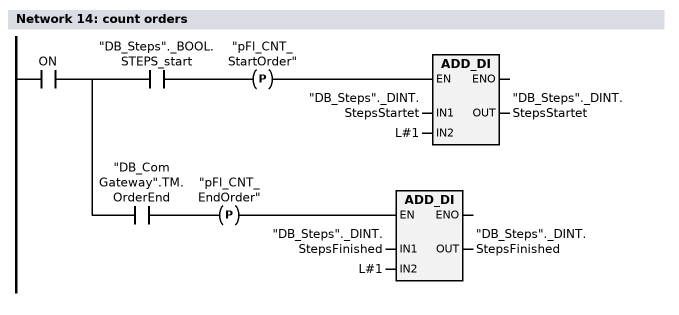
[picture p118: STEPS_OrderData networks 14-14]
NETWORK
TITLE = count orders
      A     "ON";
      =     L 35.0;
      A     L 35.0;
      A(;
      A     "DB_Steps"._BOOL.STEPS_start;
      BLD   100;
      FP    "pFl_CNT_StartOrder";
      );
      JNB   _007;
      L     "DB_Steps"._DINT.StepsStartet;
      L     L#1;
      +D;
      T     "DB_Steps"._DINT.StepsStartet;
_007: NOP   0;
      A     L 35.0;
      A(;
      A     "DB_ComGateway".TM.OrderEnd;
      BLD   100;
      FP    "pFl_CNT_EndOrder";
      );
      JNB   _008;
      L     "DB_Steps"._DINT.StepsFinished;
      L     L#1;
      +D;
      T     "DB_Steps"._DINT.StepsFinished;
_008: NOP   0;
END_FUNCTION

FUNCTION "STEPS_EMPTY" : VOID	// FC 113
TITLE = Steps Empty
VERSION : 0.1
BEGIN
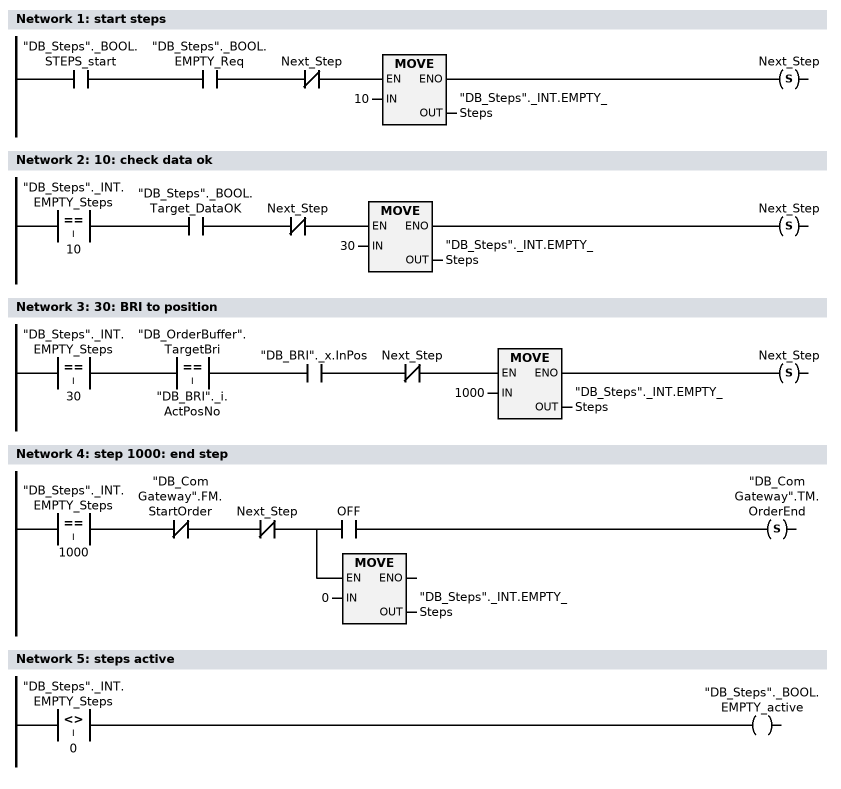
NETWORK
TITLE = start steps
      A     "DB_Steps"._BOOL.STEPS_start;
      A     "DB_Steps"._BOOL.EMPTY_Req;
      AN    "Next_Step";
      JNB   _001;
      L     10;
      T     "DB_Steps"._INT.EMPTY_Steps;
      SET;
      SAVE;
      CLR;
_001: A     BR;
      S     "Next_Step";
NETWORK
TITLE = 10: check data ok
      A(;
      L     "DB_Steps"._INT.EMPTY_Steps;
      L     10;
      ==I;
      );
      A     "DB_Steps"._BOOL.Target_DataOK;
      AN    "Next_Step";
      JNB   _002;
      L     30;
      T     "DB_Steps"._INT.EMPTY_Steps;
      SET;
      SAVE;
      CLR;
_002: A     BR;
      S     "Next_Step";
NETWORK
TITLE = 30: BRI to position
//1000: end of steps
      A(;
      L     "DB_Steps"._INT.EMPTY_Steps;
      L     30;
      ==I;
      );
      A(;
      L     "DB_OrderBuffer".TargetBri;
      L     "DB_BRI"._i.ActPosNo;
      ==I;
      );
      A     "DB_BRI"._x.InPos;
      AN    "Next_Step";
      JNB   _003;
      L     1000;
      T     "DB_Steps"._INT.EMPTY_Steps;
      SET;
      SAVE;
      CLR;
_003: A     BR;
      S     "Next_Step";
NETWORK
TITLE = step 1000: end step
//because of time reason we disable the finish flag
//also we check at the end the start bit has been cleared
      A(;
      L     "DB_Steps"._INT.EMPTY_Steps;
      L     1000;
      ==I;
      );
      AN    "DB_ComGateway".FM.StartOrder;
      AN    "Next_Step";
      =     L 0.0;
      A     L 0.0;
      A     "OFF";
      S     "DB_ComGateway".TM.OrderEnd;
      A     L 0.0;
      JNB   _004;
      L     0;
      T     "DB_Steps"._INT.EMPTY_Steps;
_004: NOP   0;
NETWORK
TITLE = steps active
      L     "DB_Steps"._INT.EMPTY_Steps;
      L     0;
      <>I;
      =     "DB_Steps"._BOOL.EMPTY_active;
END_FUNCTION

FUNCTION "Axis_BRIDGE" : VOID	// FC 200
TITLE = Axis BRIDGE
AUTHOR : Koenig
VERSION : 0.1
VAR_TEMP
  Signal : BOOL ;
  TEMP_01 : BOOL ;
  TEMP_02 : BOOL ;
  Encoder : DINT ;
  Temp_Dint : DINT ;
END_VAR
BEGIN
NETWORK
TITLE =
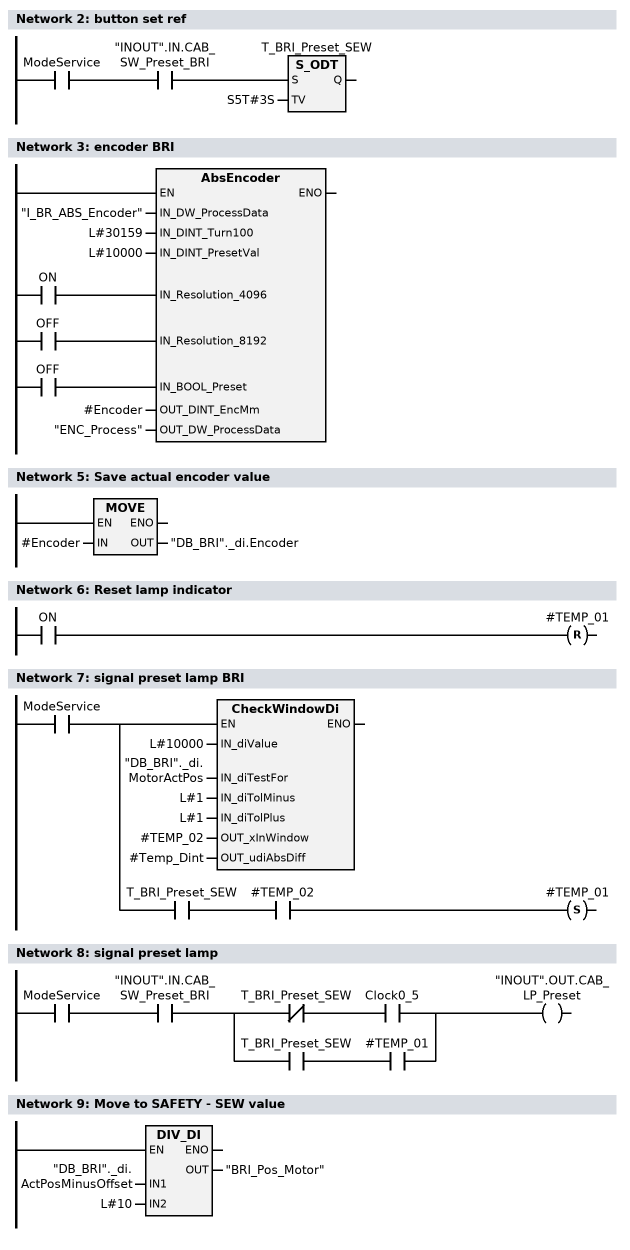
NETWORK
TITLE = button set ref
      A     "ModeService";
      A     "INOUT".IN.CAB_SW_Preset_BRI;
      L     S5T#3S;
      SD    "T_BRI_Preset_SEW";
      NOP   0;
      NOP   0;
      NOP   0;
      NOP   0;
NETWORK
TITLE = encoder BRI
      A     "ON";
      =     L 10.0;
      BLD   103;
      A     "OFF";
      =     L 10.1;
      BLD   103;
      A     "OFF";
      =     L 10.2;
      BLD   103;
      CALL  "AbsEncoder" (
           IN_DW_ProcessData        := "I_BR_ABS_Encoder",
           IN_DINT_Turn100          := L#30159,
           IN_DINT_PresetVal        := L#10000,
           IN_Resolution_4096       := L 10.0,
           IN_Resolution_8192       := L 10.1,
           IN_BOOL_Preset           := L 10.2,
           OUT_DINT_EncMm           := #Encoder,
           OUT_DW_ProcessData       := "ENC_Process");
      NOP   0;
NETWORK
TITLE = Preset encoder T&R
      A     "T_BRI_Preset_SEW";
      =     L 10.0;
      BLD   103;
      BLD   9;
      =     L 15.0;
      CDB;
      OPN   DI 50;
      TAR2  LD 11;
      A     L 10.0;
      =     DIX 0.0;
      L     L#2038;
      T     DID 2;
      L     2;
      T     DIW 6;
      L     4;
      T     DIW 8;
      L     W#16#1002;
      T     DIW 16;
      L     4;
      T     DIW 18;
      L     0;
      T     DIW 20;
      L     P#M 84.0;
      T     DID 22;
      LAR2  P#DBX 0.0;
      UC    "WRREC";
      LAR2  LD 11;
      CDB;
      BLD   10;
      NOP   0;
NETWORK
TITLE = Save actual encoder value
      L     #Encoder;
      T     "DB_BRI"._di.Encoder;
      NOP   0;
NETWORK
TITLE = Reset lamp indicator
      A     "ON";
      R     #TEMP_01;
NETWORK
TITLE = signal preset lamp BRI
      A     "ModeService";
      =     L 10.0;
      A     L 10.0;
      JNB   _001;
      CALL  "CheckWindowDi" (
           IN_diValue               := L#10000,
           IN_diTestFor             := "DB_BRI"._di.MotorActPos,
           IN_diTolMinus            := L#1,
           IN_diTolPlus             := L#1,
           OUT_xInWindow            := #TEMP_02,
           OUT_udiAbsDiff           := #Temp_Dint);
_001: NOP   0;
      A     L 10.0;
      A     "T_BRI_Preset_SEW";
      A     #TEMP_02;
      S     #TEMP_01;
NETWORK
TITLE = signal preset lamp
      A     "ModeService";
      A     "INOUT".IN.CAB_SW_Preset_BRI;
      A(;
      AN    "T_BRI_Preset_SEW";
      A     "Clock0_5";
      O;
      A     "T_BRI_Preset_SEW";
      A     #TEMP_01;
      );
      =     "INOUT".OUT.CAB_LP_Preset;
NETWORK
TITLE = Move to SAFETY - SEW value
      L     "DB_BRI"._di.ActPosMinusOffset;
      L     L#10;
      /D;
      T     "BRI_Pos_Motor";
      NOP   0;
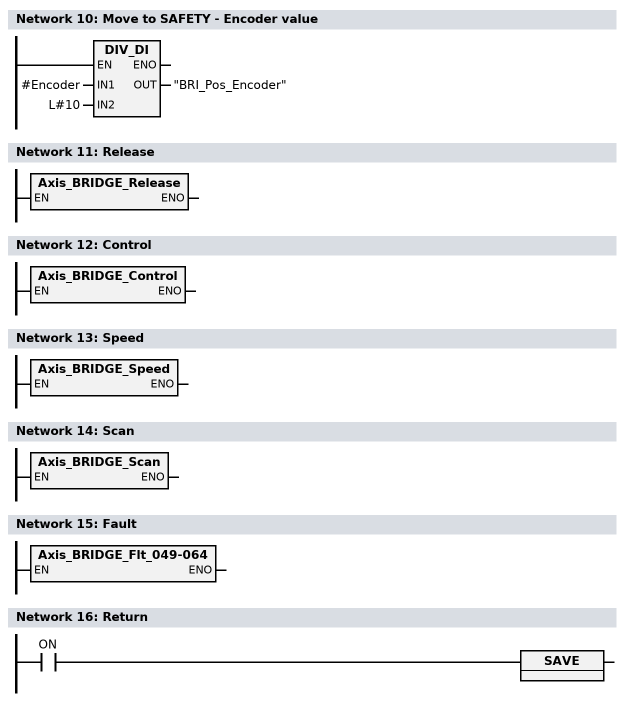
NETWORK
TITLE = Move to SAFETY - Encoder value
      L     #Encoder;
      L     L#10;
      /D;
      T     "BRI_Pos_Encoder";
      NOP   0;
NETWORK
TITLE = Release
      CALL  "Axis_BRIDGE_Release";
      NOP   0;
NETWORK
TITLE = Control
      CALL  "Axis_BRIDGE_Control";
      NOP   0;
NETWORK
TITLE = Speed
      CALL  "Axis_BRIDGE_Speed";
      NOP   0;
NETWORK
TITLE = Scan
      CALL  "Axis_BRIDGE_Scan";
      NOP   0;
NETWORK
TITLE = Fault
      CALL  "Axis_BRIDGE_Flt_049-064";
      NOP   0;
NETWORK
TITLE = Return
      A     "ON";
      SAVE;
END_FUNCTION

FUNCTION "Axis_BRIDGE_Release" : VOID	// FC 201
TITLE = Axis BRIDGE Release
VERSION : 0.1
BEGIN
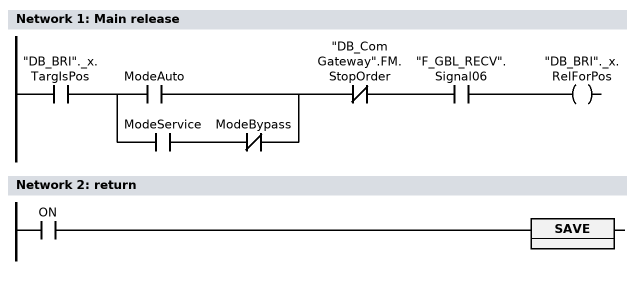
NETWORK
TITLE = Main release
      A     "DB_BRI"._x.TargIsPos;
      A(;
      O     "ModeAuto";
      O;
      A     "ModeService";
      AN    "ModeBypass";
      );
      AN    "DB_ComGateway".FM.StopOrder;
      A     "F_GBL_RECV".Signal06;
      =     "DB_BRI"._x.RelForPos;
NETWORK
TITLE = return
      A     "ON";
      SAVE;
END_FUNCTION

FUNCTION "Axis_BRIDGE_Control" : VOID	// FC 202
TITLE = BRIDGE Control
VERSION : 0.1
VAR_TEMP
  PositionMode : BOOL ;
  tmp_TagetPos_Auto : BOOL ;
  tmp_TagetPos_Manual : BOOL ;
  tmp_TargetValueOK : BOOL ;
  Mode_ref : BOOL ;
  Mode_jog : BOOL ;
  Error : WORD ;
  Next : DINT ;
  Prev : DINT ;
  First : DINT ;
  Last : DINT ;
END_VAR
BEGIN
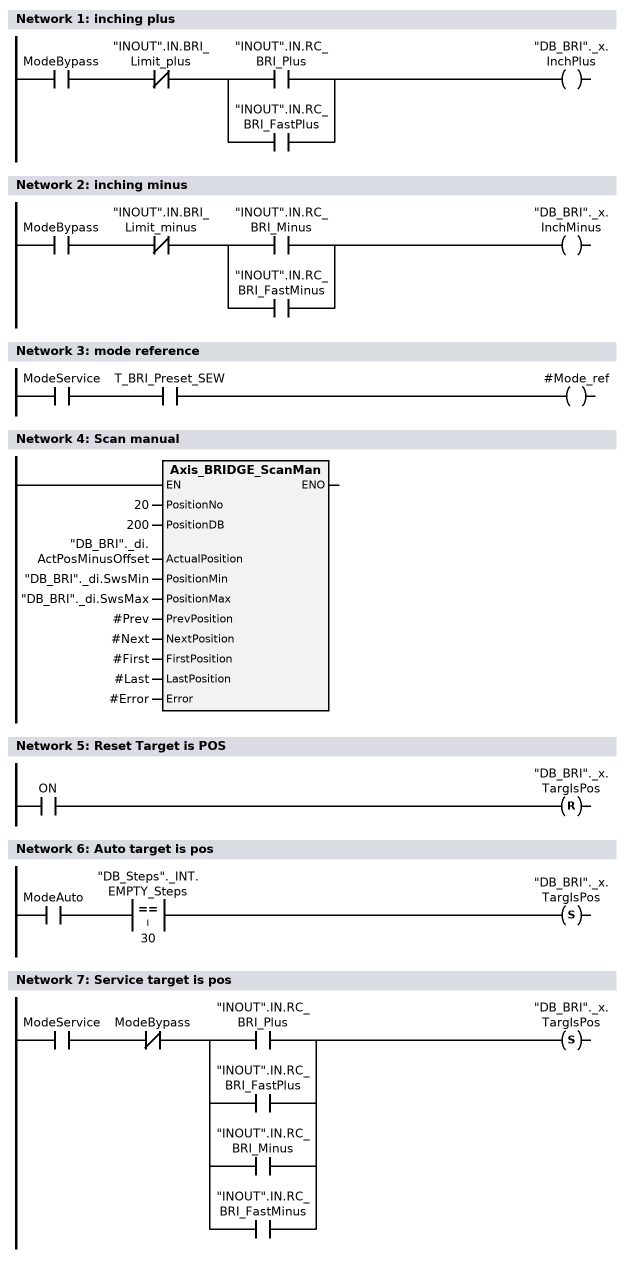
NETWORK
TITLE = inching plus
//in Service with bypass we use jog mode
      A     "ModeBypass";
      AN    "INOUT".IN.BRI_Limit_plus;
      A(;
      O     "INOUT".IN.RC_BRI_Plus;
      O     "INOUT".IN.RC_BRI_FastPlus;
      );
      =     "DB_BRI"._x.InchPlus;
NETWORK
TITLE = inching minus
      A     "ModeBypass";
      AN    "INOUT".IN.BRI_Limit_minus;
      A(;
      O     "INOUT".IN.RC_BRI_Minus;
      O     "INOUT".IN.RC_BRI_FastMinus;
      );
      =     "DB_BRI"._x.InchMinus;
NETWORK
TITLE = mode reference
      A     "ModeService";
      A     "T_BRI_Preset_SEW";
      =     #Mode_ref;
NETWORK
TITLE = Scan manual
      CALL  "Axis_BRIDGE_ScanMan" (
           PositionNo               := 20,
           PositionDB               := 200,
           ActualPosition           := "DB_BRI"._di.ActPosMinusOffset,
           PositionMin              := "DB_BRI"._di.SwsMin,
           PositionMax              := "DB_BRI"._di.SwsMax,
           PrevPosition             := #Prev,
           NextPosition             := #Next,
           FirstPosition            := #First,
           LastPosition             := #Last,
           Error                    := #Error);
      NOP   0;
NETWORK
TITLE = Reset Target is POS
      A     "ON";
      R     "DB_BRI"._x.TargIsPos;
NETWORK
TITLE = Auto target is pos
      A     "ModeAuto";
      A(;
      L     "DB_Steps"._INT.EMPTY_Steps;
      L     30;
      ==I;
      );
      S     "DB_BRI"._x.TargIsPos;
NETWORK
TITLE = Service target is pos
      A     "ModeService";
      AN    "ModeBypass";
      A(;
      O     "INOUT".IN.RC_BRI_Plus;
      O     "INOUT".IN.RC_BRI_FastPlus;
      O     "INOUT".IN.RC_BRI_Minus;
      O     "INOUT".IN.RC_BRI_FastMinus;
      );
      S     "DB_BRI"._x.TargIsPos;
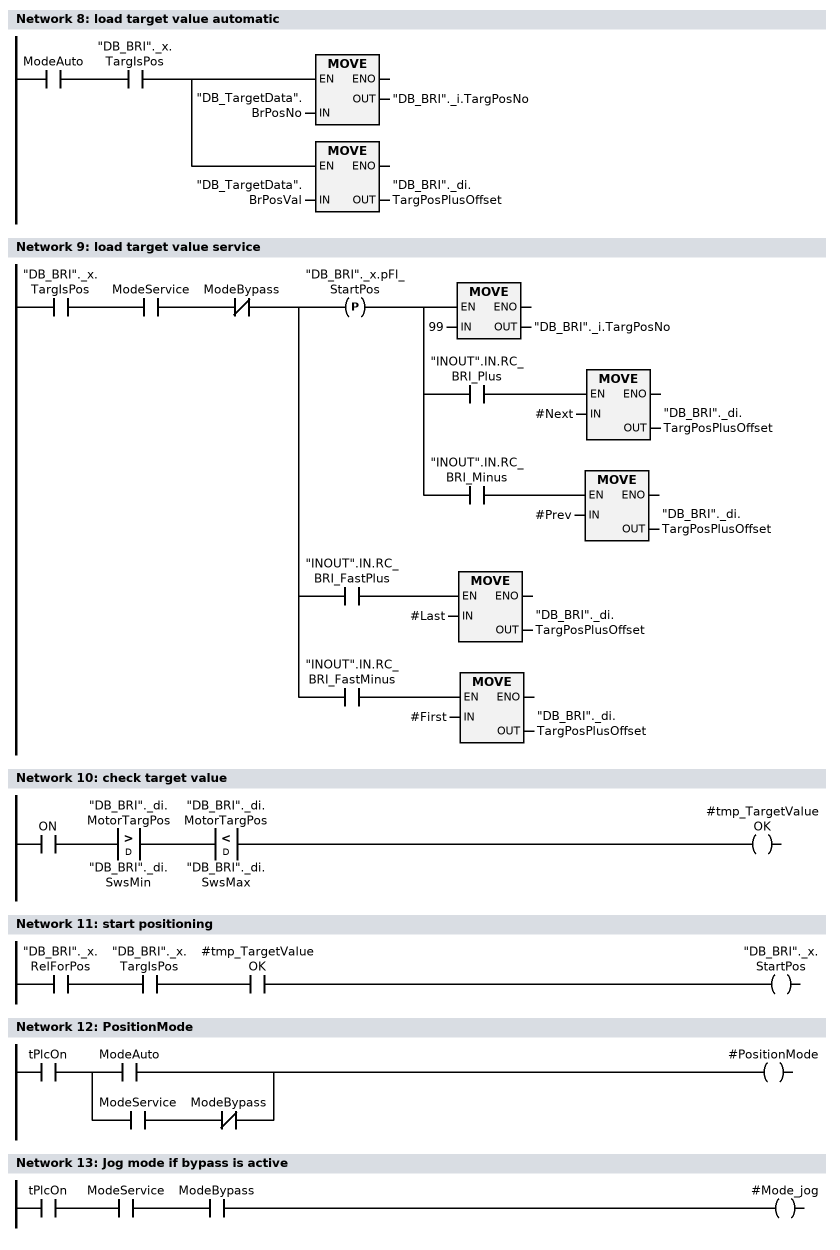
NETWORK
TITLE = load target value automatic
      A     "ModeAuto";
      A     "DB_BRI"._x.TargIsPos;
      =     L 20.0;
      A     L 20.0;
      JNB   _001;
      L     "DB_TargetData".BrPosNo;
      T     "DB_BRI"._i.TargPosNo;
_001: NOP   0;
      A     L 20.0;
      JNB   _002;
      L     "DB_TargetData".BrPosVal;
      T     "DB_BRI"._di.TargPosPlusOffset;
_002: NOP   0;
NETWORK
TITLE = load target value service
//In service we load the next/prev value or min/max
      A     "DB_BRI"._x.TargIsPos;
      A     "ModeService";
      AN    "ModeBypass";
      =     L 20.0;
      A     L 20.0;
      FP    "DB_BRI"._x.pFl_StartPos;
      =     L 20.1;
      A     L 20.1;
      JNB   _003;
      L     99;
      T     "DB_BRI"._i.TargPosNo;
_003: NOP   0;
      A     L 20.1;
      A     "INOUT".IN.RC_BRI_Plus;
      JNB   _004;
      L     #Next;
      T     "DB_BRI"._di.TargPosPlusOffset;
_004: NOP   0;
      A     L 20.1;
      A     "INOUT".IN.RC_BRI_Minus;
      JNB   _005;
      L     #Prev;
      T     "DB_BRI"._di.TargPosPlusOffset;
_005: NOP   0;
      A     L 20.0;
      A     "INOUT".IN.RC_BRI_FastPlus;
      JNB   _006;
      L     #Last;
      T     "DB_BRI"._di.TargPosPlusOffset;
_006: NOP   0;
      A     L 20.0;
      A     "INOUT".IN.RC_BRI_FastMinus;
      JNB   _007;
      L     #First;
      T     "DB_BRI"._di.TargPosPlusOffset;
_007: NOP   0;
NETWORK
TITLE = check target value
      A     "ON";
      A(;
      L     "DB_BRI"._di.MotorTargPos;
      L     "DB_BRI"._di.SwsMin;
      >D;
      );
      A(;
      L     "DB_BRI"._di.MotorTargPos;
      L     "DB_BRI"._di.SwsMax;
      <D;
      );
      =     #tmp_TargetValueOK;
NETWORK
TITLE = start positioning
      A     "DB_BRI"._x.RelForPos;
      A     "DB_BRI"._x.TargIsPos;
      A     #tmp_TargetValueOK;
      =     "DB_BRI"._x.StartPos;
NETWORK
TITLE = PositionMode
      A     "tPlcOn";
      A(;
      O     "ModeAuto";
      O;
      A     "ModeService";
      AN    "ModeBypass";
      );
      =     #PositionMode;
NETWORK
TITLE = Jog mode if bypass is active
      A     "tPlcOn";
      A     "ModeService";
      A     "ModeBypass";
      =     #Mode_jog;
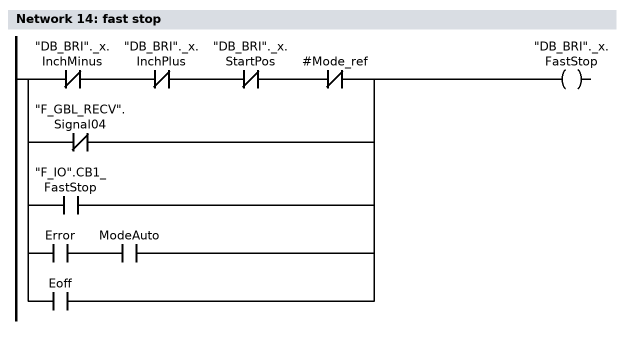
NETWORK
TITLE = fast stop
      AN    "DB_BRI"._x.InchMinus;
      AN    "DB_BRI"._x.InchPlus;
      AN    "DB_BRI"._x.StartPos;
      AN    #Mode_ref;
      ON    "F_GBL_RECV".Signal04;
      O     "F_IO".CB1_FastStop;
      O;
      A     "Error";
      A     "ModeAuto";
      O     "Eoff";
      =     "DB_BRI"._x.FastStop;
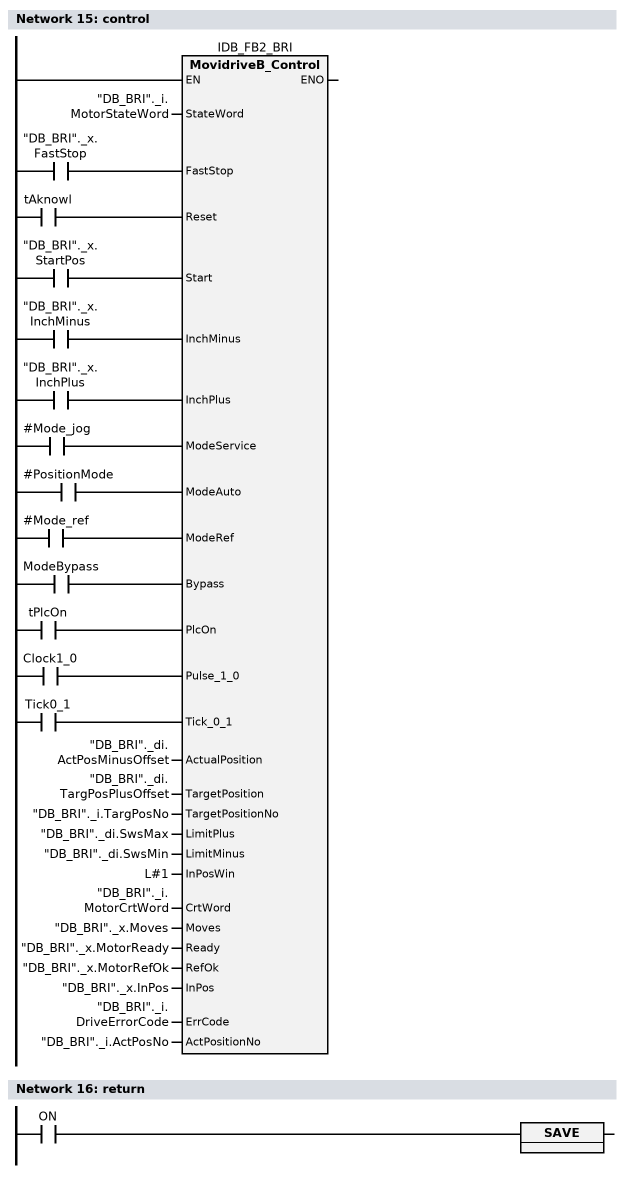
NETWORK
TITLE = control
      A     "DB_BRI"._x.FastStop;
      =     L 20.0;
      BLD   103;
      A     "tAknowl";
      =     L 20.1;
      BLD   103;
      A     "DB_BRI"._x.StartPos;
      =     L 20.2;
      BLD   103;
      A     "DB_BRI"._x.InchMinus;
      =     L 20.3;
      BLD   103;
      A     "DB_BRI"._x.InchPlus;
      =     L 20.4;
      BLD   103;
      A     #Mode_jog;
      =     L 20.5;
      BLD   103;
      A     #PositionMode;
      =     L 20.6;
      BLD   103;
      A     #Mode_ref;
      =     L 20.7;
      BLD   103;
      A     "ModeBypass";
      =     L 21.0;
      BLD   103;
      A     "tPlcOn";
      =     L 21.1;
      BLD   103;
      A     "Clock1_0";
      =     L 21.2;
      BLD   103;
      A     "Tick0_1";
      =     L 21.3;
      BLD   103;
      CALL  "MovidriveB_Control" , "IDB_FB2_BRI" (
           StateWord                := "DB_BRI"._i.MotorStateWord,
           FastStop                 := L 20.0,
           Reset                    := L 20.1,
           Start                    := L 20.2,
           InchMinus                := L 20.3,
           InchPlus                 := L 20.4,
           ModeService              := L 20.5,
           ModeAuto                 := L 20.6,
           ModeRef                  := L 20.7,
           Bypass                   := L 21.0,
           PlcOn                    := L 21.1,
           Pulse_1_0                := L 21.2,
           Tick_0_1                 := L 21.3,
           ActualPosition           := "DB_BRI"._di.ActPosMinusOffset,
           TargetPosition           := "DB_BRI"._di.TargPosPlusOffset,
           TargetPositionNo         := "DB_BRI"._i.TargPosNo,
           LimitPlus                := "DB_BRI"._di.SwsMax,
           LimitMinus               := "DB_BRI"._di.SwsMin,
           InPosWin                 := L#1,
           CrtWord                  := "DB_BRI"._i.MotorCrtWord,
           Moves                    := "DB_BRI"._x.Moves,
           Ready                    := "DB_BRI"._x.MotorReady,
           RefOk                    := "DB_BRI"._x.MotorRefOk,
           InPos                    := "DB_BRI"._x.InPos,
           ErrCode                  := "DB_BRI"._i.DriveErrorCode,
           ActPositionNo            := "DB_BRI"._i.ActPosNo);
      NOP   0;
NETWORK
TITLE = return
      A     "ON";
      SAVE;
END_FUNCTION

FUNCTION "Axis_BRIDGE_Speed" : VOID	// FC 203
TITLE = BRIDGE Speed
VERSION : 0.1
VAR_TEMP
  tmp_di_1 : DINT ;
  tmp_di_2 : DINT ;
  tmp_i_1 : INT ;
  tmp_i_2 : INT ;
  tmp_speed : INT ;
  tmp_diff_Pos : DINT ;
  tmp_Slow_Pos : BOOL ;
  tmp_Dcc : INT ;
END_VAR
BEGIN
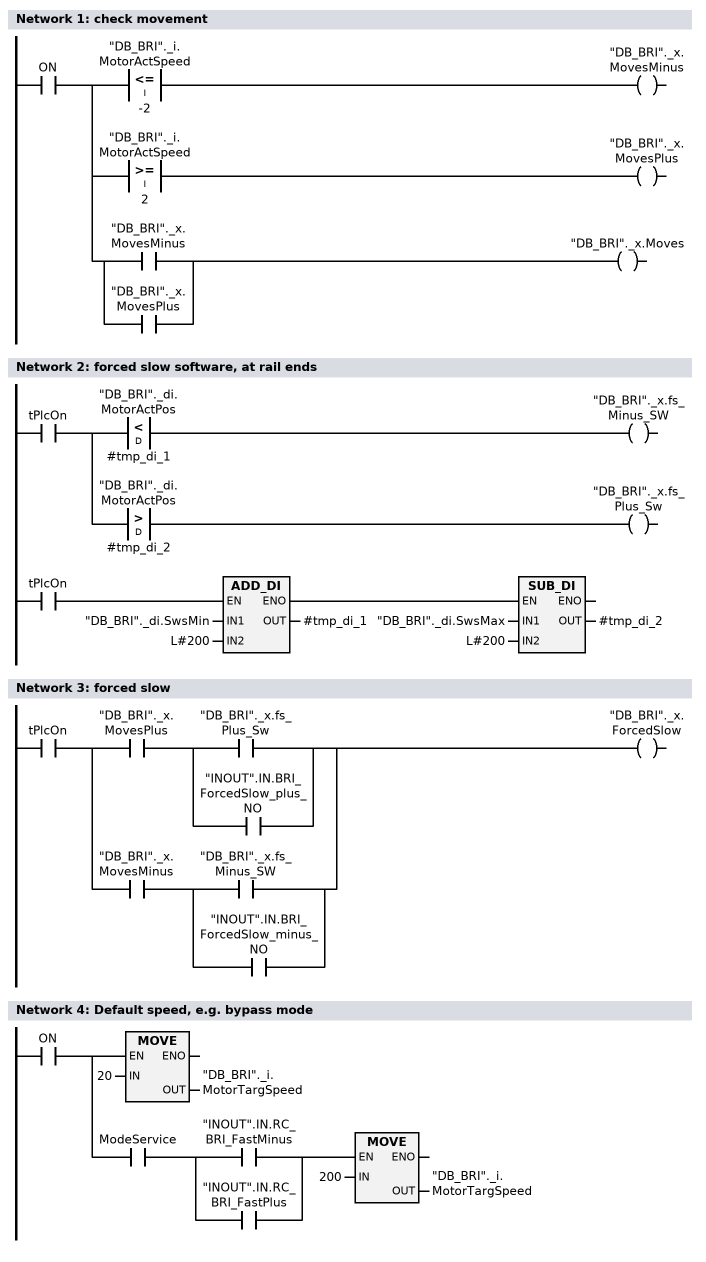
NETWORK
TITLE = check movement
      A     "ON";
      =     L 22.0;
      A     L 22.0;
      A(;
      L     "DB_BRI"._i.MotorActSpeed;
      L     -2;
      <=I;
      );
      =     "DB_BRI"._x.MovesMinus;
      A     L 22.0;
      A(;
      L     "DB_BRI"._i.MotorActSpeed;
      L     2;
      >=I;
      );
      =     "DB_BRI"._x.MovesPlus;
      A     L 22.0;
      A(;
      O     "DB_BRI"._x.MovesMinus;
      O     "DB_BRI"._x.MovesPlus;
      );
      =     "DB_BRI"._x.Moves;
NETWORK
TITLE = forced slow software, at rail ends
//Old distance: 1000mm
      A     "tPlcOn";
      =     L 22.0;
      A(;
      A     L 22.0;
      JNB   _001;
      L     "DB_BRI"._di.SwsMin;
      L     L#200;
      +D;
      T     #tmp_di_1;
      AN    OV;
      SAVE;
      CLR;
_001: A     BR;
      );
      JNB   _002;
      L     "DB_BRI"._di.SwsMax;
      L     L#200;
      -D;
      T     #tmp_di_2;
_002: NOP   0;
      A     L 22.0;
      A(;
      L     "DB_BRI"._di.MotorActPos;
      L     #tmp_di_1;
      <D;
      );
      =     "DB_BRI"._x.fs_Minus_SW;
      A     L 22.0;
      A(;
      L     "DB_BRI"._di.MotorActPos;
      L     #tmp_di_2;
      >D;
      );
      =     "DB_BRI"._x.fs_Plus_Sw;
NETWORK
TITLE = forced slow
//in service we use only the software, in auto we use the prox. switches
      A     "tPlcOn";
      A(;
      A     "DB_BRI"._x.MovesPlus;
      A(;
      O     "DB_BRI"._x.fs_Plus_Sw;
      O     "INOUT".IN.BRI_ForcedSlow_plus_NO;
      );
      O;
      A     "DB_BRI"._x.MovesMinus;
      A(;
      O     "DB_BRI"._x.fs_Minus_SW;
      O     "INOUT".IN.BRI_ForcedSlow_minus_NO;
      );
      );
      =     "DB_BRI"._x.ForcedSlow;
NETWORK
TITLE = Default speed, e.g. bypass mode
//in bypass we can also drive a little faster
//
      A     "ON";
      =     L 22.0;
      A     L 22.0;
      JNB   _003;
      L     20;
      T     "DB_BRI"._i.MotorTargSpeed;
_003: NOP   0;
      A     L 22.0;
      A     "ModeService";
      A(;
      O     "INOUT".IN.RC_BRI_FastMinus;
      O     "INOUT".IN.RC_BRI_FastPlus;
      );
      JNB   _004;
      L     200;
      T     "DB_BRI"._i.MotorTargSpeed;
_004: NOP   0;
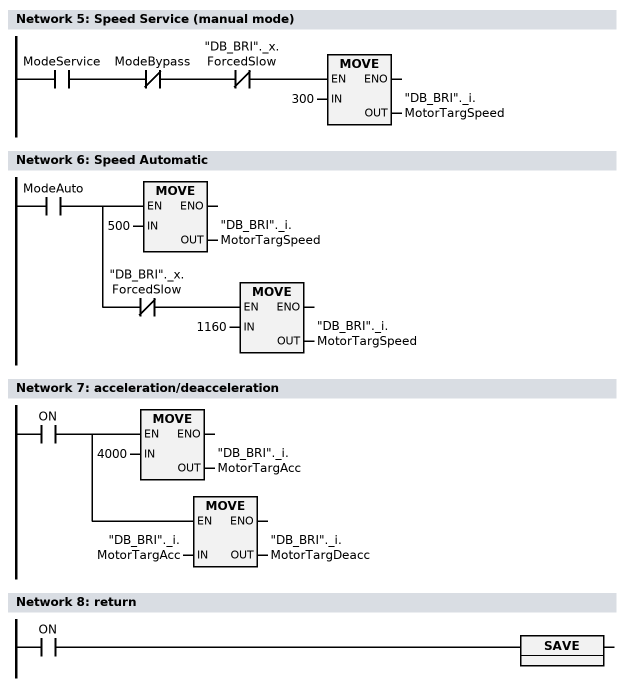
NETWORK
TITLE = Speed Service (manual mode)
//in bypass we do not allow faster speed
//Speed fast old: 200
      A     "ModeService";
      AN    "ModeBypass";
      AN    "DB_BRI"._x.ForcedSlow;
      JNB   _005;
      L     300;
      T     "DB_BRI"._i.MotorTargSpeed;
_005: NOP   0;
NETWORK
TITLE = Speed Automatic
//70m/min max
//1,16 m/s
      A     "ModeAuto";
      =     L 22.0;
      A     L 22.0;
      JNB   _006;
      L     500;
      T     "DB_BRI"._i.MotorTargSpeed;
_006: NOP   0;
      A     L 22.0;
      AN    "DB_BRI"._x.ForcedSlow;
      JNB   _007;
      L     1160;
      T     "DB_BRI"._i.MotorTargSpeed;
_007: NOP   0;
NETWORK
TITLE = acceleration/deacceleration
//0,45 m/S2
//2.6 s
      A     "ON";
      =     L 22.0;
      A     L 22.0;
      JNB   _008;
      L     4000;
      T     "DB_BRI"._i.MotorTargAcc;
_008: NOP   0;
      A     L 22.0;
      JNB   _009;
      L     "DB_BRI"._i.MotorTargAcc;
      T     "DB_BRI"._i.MotorTargDeacc;
_009: NOP   0;
NETWORK
TITLE = return
      A     "ON";
      SAVE;
END_FUNCTION

FUNCTION "Axis_BRIDGE_Scan" : VOID	// FC 204
TITLE = BRIDGE Scan
VERSION : 0.1
VAR_TEMP
  tmp_di_1 : DINT ;
  tmp_di_PosWin : DINT ;
  tmp_i_BRIScanSetNo : INT ;
  tmp_i_LIF_DBNo : INT ;
  tmp_i_LIF_DBNo_2 : INT ;
  tmp_di_Scan_Plus : DINT ;
  tmp_di_Scan_Minus : DINT ;
  tmp_di_Scan_Pos : DINT ;
  tmp_di_Bri_Pos : DINT ;
  tmp_db_no : INT ;
END_VAR
BEGIN
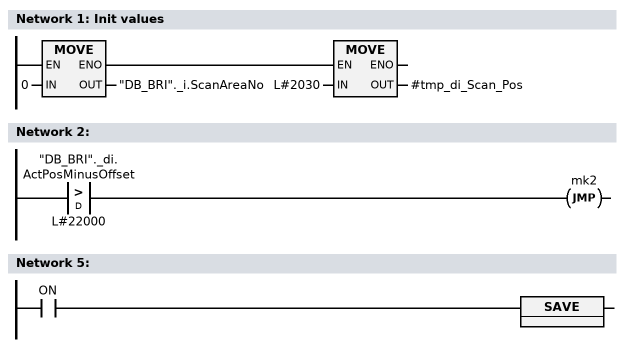
NETWORK
TITLE = Init values
      A(;
      L     0;
      T     "DB_BRI"._i.ScanAreaNo;
      SET;
      SAVE;
      CLR;
      A     BR;
      );
      JNB   _001;
      L     L#2030;
      T     #tmp_di_Scan_Pos;
_001: NOP   0;
NETWORK
TITLE =
      L     "DB_BRI"._di.ActPosMinusOffset;
      L     L#22000;
      >D;
      JC    mk2;
NETWORK
TITLE = Calculating the Bridge Scan area
//for display on remote
      L     "DB_BRI"._di.ActPosMinusOffset;
      L     L#3900;
      -D;
      DTR;
      L     3.050000e+03;
      /R;
      RND;
      L     11;	// turn value
      TAK;
      -I;
      T     "DB_BRI"._i.ScanAreaNo;
      JU    mk;
NETWORK
TITLE = Calculating the Bridge Scan area
//for display on remote
mk2:  L     "DB_BRI"._di.ActPosMinusOffset;
      L     L#6400;
      -D;
      DTR;
      L     3.050000e+03;
      /R;
      RND;
      L     11;	// turn value
      TAK;
      -I;
      T     "DB_BRI"._i.ScanAreaNo;
NETWORK
TITLE =
mk:   A     "ON";
      SAVE;
END_FUNCTION

FUNCTION "Axis_BRIDGE_ScanMan" : VOID	// FC 205
TITLE = Scan manual pos
//
//Baustein-Kommentar ...
//
AUTHOR : Koenig
FAMILY : Scan
NAME : ManPos
VERSION : 1.0
VAR_INPUT
  PositionNo : INT ;	//Positions number
  PositionDB : INT ;	//DB Number of Positions
  ActualPosition : DINT ;
  PositionMin : DINT ;
  PositionMax : DINT ;
END_VAR
VAR_OUTPUT
  PrevPosition : DINT ;
  NextPosition : DINT ;
  FirstPosition : DINT ;
  LastPosition : DINT ;
  Error : WORD ;
END_VAR
VAR_TEMP
  i : INT ;
  value : DINT ;
  diff : DINT ;
  DB_No : WORD ;
  DB_Length : WORD ;
  DB_WP : BOOL ;
  RETURN_Value : INT ;
END_VAR
BEGIN
// body was compiled from an SCL source; compiled code not shown
END_FUNCTION

FUNCTION "Axis_BRIDGE_Flt_049-064" : VOID	// FC 209
TITLE = Error bridge
VERSION : 0.1
BEGIN
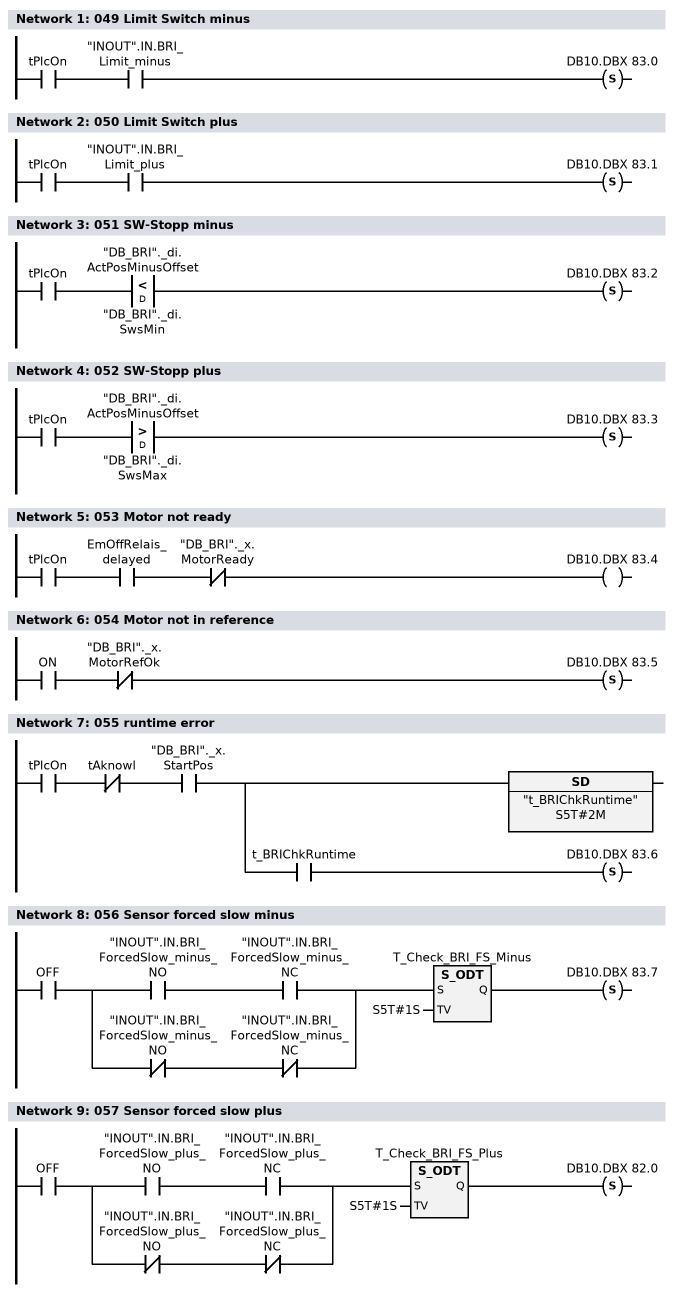
NETWORK
TITLE = 049 Limit Switch minus
      A     "tPlcOn";
      A     "INOUT".IN.BRI_Limit_minus;
      S     DB10.DBX 83.0;
NETWORK
TITLE = 050 Limit Switch plus
      A     "tPlcOn";
      A     "INOUT".IN.BRI_Limit_plus;
      S     DB10.DBX 83.1;
NETWORK
TITLE = 051 SW-Stopp minus
      A     "tPlcOn";
      A(;
      L     "DB_BRI"._di.ActPosMinusOffset;
      L     "DB_BRI"._di.SwsMin;
      <D;
      );
      S     DB10.DBX 83.2;
NETWORK
TITLE = 052 SW-Stopp plus
      A     "tPlcOn";
      A(;
      L     "DB_BRI"._di.ActPosMinusOffset;
      L     "DB_BRI"._di.SwsMax;
      >D;
      );
      S     DB10.DBX 83.3;
NETWORK
TITLE = 053 Motor not ready
      A     "tPlcOn";
      A     "EmOffRelais_delayed";
      AN    "DB_BRI"._x.MotorReady;
      =     DB10.DBX 83.4;
NETWORK
TITLE = 054 Motor not in reference
      A     "ON";
      AN    "DB_BRI"._x.MotorRefOk;
      S     DB10.DBX 83.5;
NETWORK
TITLE = 055 runtime error
      A     "tPlcOn";
      AN    "tAknowl";
      A     "DB_BRI"._x.StartPos;
      =     L 0.0;
      A     L 0.0;
      BLD   102;
      L     S5T#2M;
      SD    "t_BRIChkRuntime";
      A     L 0.0;
      A     "t_BRIChkRuntime";
      S     DB10.DBX 83.6;
NETWORK
TITLE = 056 Sensor forced slow minus
      A     "OFF";
      A(;
      A     "INOUT".IN.BRI_ForcedSlow_minus_NO;
      A     "INOUT".IN.BRI_ForcedSlow_minus_NC;
      O;
      AN    "INOUT".IN.BRI_ForcedSlow_minus_NO;
      AN    "INOUT".IN.BRI_ForcedSlow_minus_NC;
      );
      L     S5T#1S;
      SD    "T_Check_BRI_FS_Minus";
      NOP   0;
      NOP   0;
      NOP   0;
      A     "T_Check_BRI_FS_Minus";
      S     DB10.DBX 83.7;
NETWORK
TITLE = 057 Sensor forced slow plus
      A     "OFF";
      A(;
      A     "INOUT".IN.BRI_ForcedSlow_plus_NO;
      A     "INOUT".IN.BRI_ForcedSlow_plus_NC;
      O;
      AN    "INOUT".IN.BRI_ForcedSlow_plus_NO;
      AN    "INOUT".IN.BRI_ForcedSlow_plus_NC;
      );
      L     S5T#1S;
      SD    "T_Check_BRI_FS_Plus";
      NOP   0;
      NOP   0;
      NOP   0;
      A     "T_Check_BRI_FS_Plus";
      S     DB10.DBX 82.0;
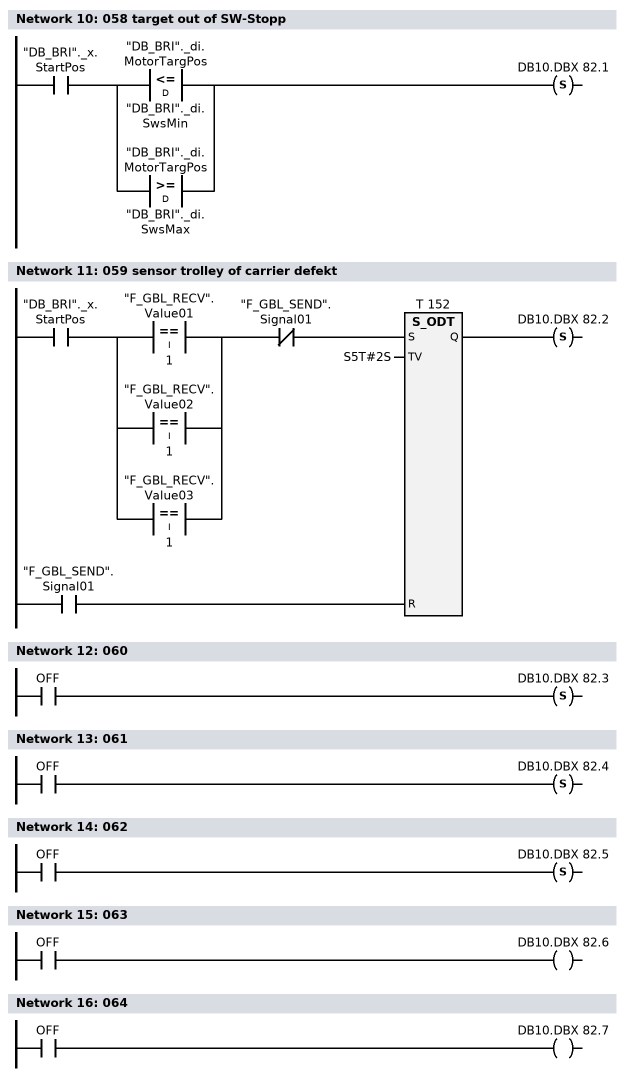
NETWORK
TITLE = 058 target out of SW-Stopp
      A     "DB_BRI"._x.StartPos;
      A(;
      O(;
      L     "DB_BRI"._di.MotorTargPos;
      L     "DB_BRI"._di.SwsMin;
      <=D;
      );
      O(;
      L     "DB_BRI"._di.MotorTargPos;
      L     "DB_BRI"._di.SwsMax;
      >=D;
      );
      );
      S     DB10.DBX 82.1;
NETWORK
TITLE = 059 sensor trolley of carrier defekt
      A     "DB_BRI"._x.StartPos;
      A(;
      O(;
      L     "F_GBL_RECV".Value01;
      L     1;
      ==I;
      );
      O(;
      L     "F_GBL_RECV".Value02;
      L     1;
      ==I;
      );
      O(;
      L     "F_GBL_RECV".Value03;
      L     1;
      ==I;
      );
      );
      AN    "F_GBL_SEND".Signal01;
      L     S5T#2S;
      SD    T 152;
      A     "F_GBL_SEND".Signal01;
      R     T 152;
      NOP   0;
      NOP   0;
      A     T 152;
      S     DB10.DBX 82.2;
NETWORK
TITLE = 060
      A     "OFF";
      S     DB10.DBX 82.3;
NETWORK
TITLE = 061
      A     "OFF";
      S     DB10.DBX 82.4;
NETWORK
TITLE = 062
      A     "OFF";
      S     DB10.DBX 82.5;
NETWORK
TITLE = 063
      A     "OFF";
      =     DB10.DBX 82.6;
NETWORK
TITLE = 064
      A     "OFF";
      =     DB10.DBX 82.7;
END_FUNCTION

FUNCTION "iPar_ServerCall" : VOID	// FC 900
VERSION : 0.1
VAR_TEMP
  tmp_date : DATE ;
  tmp_TOD : TIME_OF_DAY ;
  OB1_DATE_TIME : DATE_AND_TIME ;	//Date and time OB1 started
  on : BOOL ;
END_VAR
BEGIN
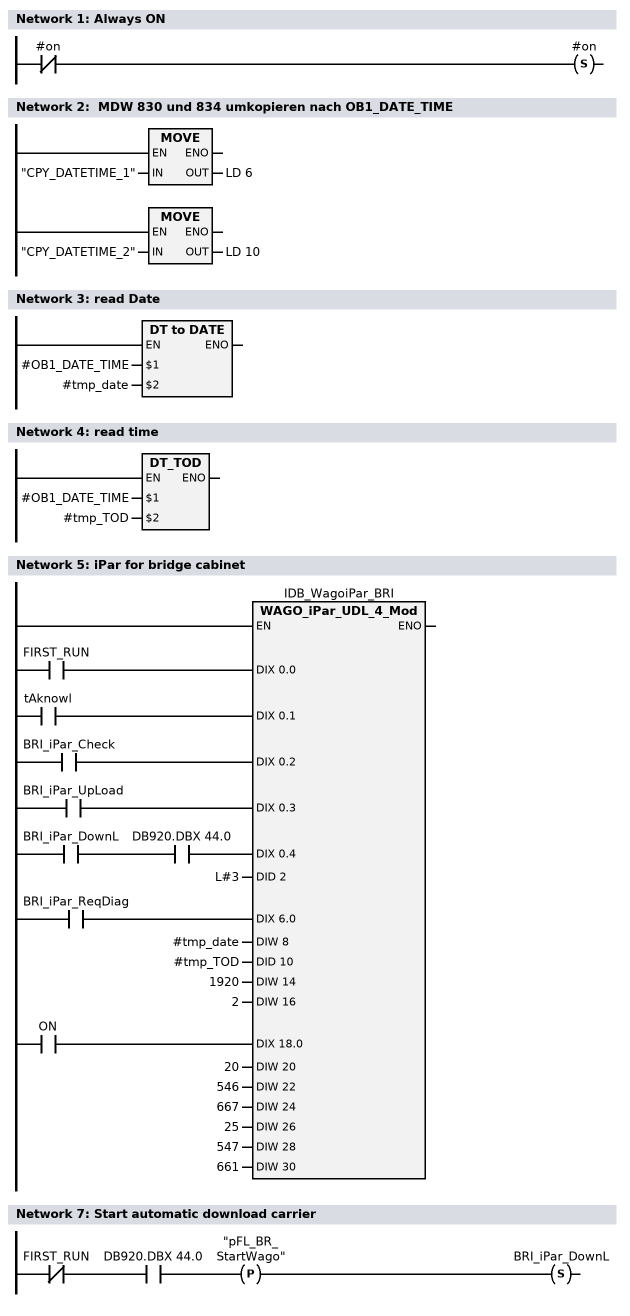
NETWORK
TITLE = Always ON
      AN    #on;
      S     #on;
NETWORK
TITLE =  MDW 830 und 834 umkopieren nach OB1_DATE_TIME
      L     "CPY_DATETIME_1";
      T     LD 6;
      L     "CPY_DATETIME_2";
      T     LD 10;
NETWORK
TITLE = read Date
      CALL  "DT to DATE" (
           $1                       := #OB1_DATE_TIME,
           $2                       := #tmp_date);
      NOP   0;
NETWORK
TITLE = read time
      CALL  "DT_TOD" (
           $1                       := #OB1_DATE_TIME,
           $2                       := #tmp_TOD);
      NOP   0;
NETWORK
TITLE = iPar for bridge cabinet
      A     "FIRST_RUN";
      =     L 15.0;
      BLD   103;
      A     "tAknowl";
      =     L 15.1;
      BLD   103;
      A     "BRI_iPar_Check";
      =     L 15.2;
      BLD   103;
      A     "BRI_iPar_UpLoad";
      =     L 15.3;
      BLD   103;
      A     "BRI_iPar_DownL";
      A     DB920.DBX 44.0;
      =     L 15.4;
      BLD   103;
      A     "BRI_iPar_ReqDiag";
      =     L 15.7;
      BLD   103;
      A     "ON";
      =     L 16.0;
      BLD   103;
      CALL  "WAGO_iPar_UDL_4_Mod" , "IDB_WagoiPar_BRI" (
           DIX 0.0                  := L 15.0,
           DIX 0.1                  := L 15.1,
           DIX 0.2                  := L 15.2,
           DIX 0.3                  := L 15.3,
           DIX 0.4                  := L 15.4,
           DID 2                    := L#3,
           DIX 6.0                  := L 15.7,
           DIW 8                    := #tmp_date,
           DID 10                   := #tmp_TOD,
           DIW 14                   := 1920,
           DIW 16                   := 2,
           DIX 18.0                 := L 16.0,
           DIW 20                   := 20,
           DIW 22                   := 546,
           DIW 24                   := 667,
           DIW 26                   := 25,
           DIW 28                   := 547,
           DIW 30                   := 661);
      NOP   0;
NETWORK
TITLE = iPar Diagnose for all modules
NETWORK
TITLE = Start automatic download carrier
      AN    "FIRST_RUN";
      A     DB920.DBX 44.0;
      FP    "pFL_BR_StartWago";
      S     "BRI_iPar_DownL";
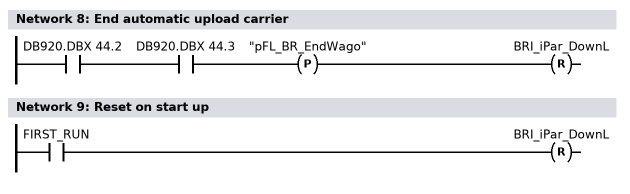
NETWORK
TITLE = End automatic upload carrier
      A     DB920.DBX 44.2;
      A     DB920.DBX 44.3;
      FP    "pFL_BR_EndWago";
      R     "BRI_iPar_DownL";
NETWORK
TITLE = Reset on start up
      A     "FIRST_RUN";
      R     "BRI_iPar_DownL";
END_FUNCTION

FUNCTION "BRIGetPosVal_New" : VOID	// FC 1071
VERSION : 0.1
VAR_INPUT
  in_x_Enable : BOOL ;
  in_i_BrPosNo : INT ;
  in_i_DBNo : INT ;
  in_i_NoOfDatasets : INT ;
  in_i_LengthDataset : INT ;
END_VAR
VAR_OUTPUT
  i_ErrCode : INT ;
  i_BrTrPosNo : INT ;
  di_BrPosVal : DINT ;
END_VAR
VAR_TEMP
  Save_AR1 : DWORD ;
  Save_AR2 : DWORD ;
  tmp_di_Pointer : DINT ;
  tmp_di_1 : DINT ;
  tmp_di_PosVal : DINT ;
  tmp_i_DBNo : INT ;
  tmp_i_ErrCode : INT ;
  tmp_i_Counter : INT ;
  tmp_i_ChkPosNo : INT ;
  tmp_i_PosNo : INT ;
  ON : BOOL ;
  tmp_x_OK : BOOL ;
END_VAR
BEGIN
NETWORK
TITLE = save register
      TAR1  #Save_AR1;
      TAR2  #Save_AR2;
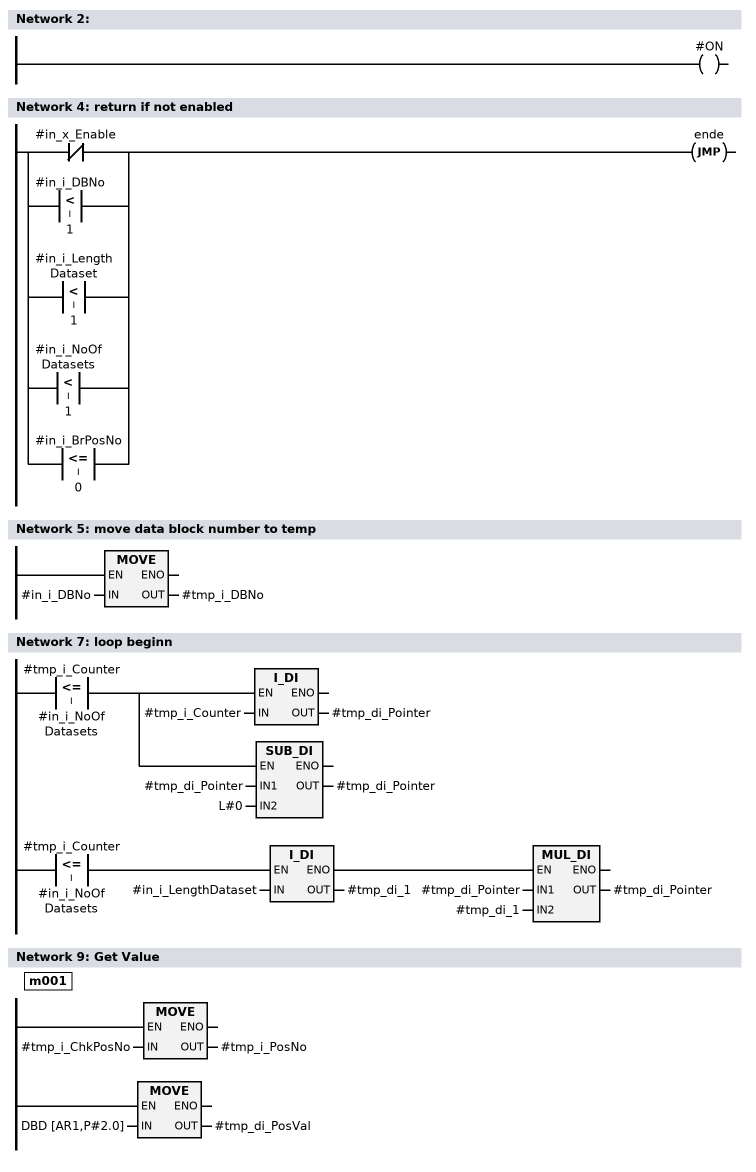
NETWORK
TITLE =
      SET;
      =     #ON;
NETWORK
TITLE = init
      L     0;
      T     #tmp_i_ErrCode;
      L     0;
      T     #tmp_i_ChkPosNo;
      L     L#0;
      T     #tmp_di_PosVal;
      L     L#0;
      T     #tmp_di_Pointer;
      L     0;
      T     #tmp_i_Counter;
      CLR;
      R     #tmp_x_OK;
NETWORK
TITLE = return if not enabled
      ON    #in_x_Enable;
      O(;
      L     #in_i_DBNo;
      L     1;
      <I;
      );
      O(;
      L     #in_i_LengthDataset;
      L     1;
      <I;
      );
      O(;
      L     #in_i_NoOfDatasets;
      L     1;
      <I;
      );
      O(;
      L     #in_i_BrPosNo;
      L     0;
      <=I;
      );
      JC    ende;
NETWORK
TITLE = move data block number to temp
      L     #in_i_DBNo;
      T     #tmp_i_DBNo;
      NOP   0;
NETWORK
TITLE = open db
      OPN   DB [#tmp_i_DBNo];
NETWORK
TITLE = loop beginn
//calculate pointer to positionvalue
scbr: L     #tmp_i_Counter;
      L     #in_i_NoOfDatasets;
      <=I;
      =     L 31.0;
      A     L 31.0;
      JNB   _001;
      L     #tmp_i_Counter;
      ITD;
      T     #tmp_di_Pointer;
_001: NOP   0;
      A     L 31.0;
      JNB   _002;
      L     #tmp_di_Pointer;
      L     L#0;
      -D;
      T     #tmp_di_Pointer;
_002: NOP   0;
      A(;
      A     L 31.0;
      JNB   _003;
      L     #in_i_LengthDataset;
      ITD;
      T     #tmp_di_1;
      SET;
      SAVE;
      CLR;
_003: A     BR;
      );
      JNB   _004;
      L     #tmp_di_Pointer;
      L     #tmp_di_1;
      *D;
      T     #tmp_di_Pointer;
_004: NOP   0;
NETWORK
TITLE =
      L     #tmp_di_Pointer;
      SLD   3;
      LAR1;
      L     DBW [AR1,P#0.0];
      T     #tmp_i_ChkPosNo;
      L     #tmp_i_ChkPosNo;
      L     #in_i_BrPosNo;
      ==I;
      JC    m001;
      L     #tmp_i_Counter;
      L     1;
      +I;
      T     #tmp_i_Counter;
      L     #tmp_i_Counter;
      L     #in_i_NoOfDatasets;
      <=I;
      JC    scbr;
      JU    ende;
NETWORK
TITLE = Get Value
m001: NOP   0;
      L     #tmp_i_ChkPosNo;
      T     #tmp_i_PosNo;
      L     DBD [AR1,P#2.0];
      T     #tmp_di_PosVal;
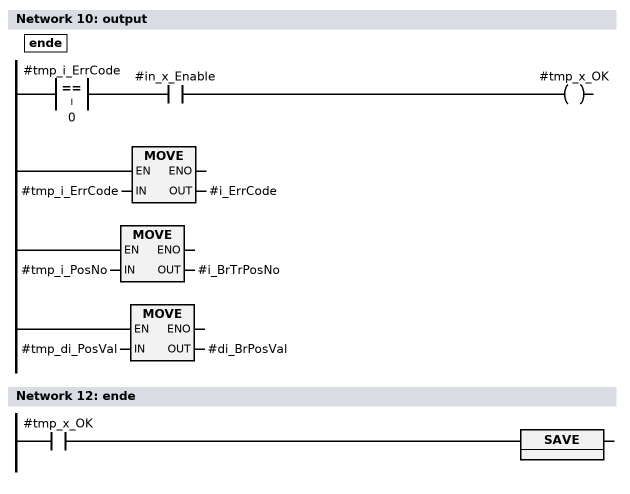
NETWORK
TITLE = output
ende: NOP   0;
      L     #tmp_i_ErrCode;
      L     0;
      ==I;
      A     #in_x_Enable;
      =     #tmp_x_OK;
      L     #tmp_i_ErrCode;
      T     #i_ErrCode;
      L     #tmp_i_PosNo;
      T     #i_BrTrPosNo;
      L     #tmp_di_PosVal;
      T     #di_BrPosVal;
NETWORK
TITLE = restore register
      LAR1  #Save_AR1;
      LAR2  #Save_AR2;
NETWORK
TITLE = ende
      A     #tmp_x_OK;
      SAVE;
END_FUNCTION

// DB 1: know-how protected block, not included

DATA_BLOCK "DB_BRI"	// DB 5
VERSION : 0.1
  STRUCT
   _di : STRUCT
    MotorTargPos : DINT ;
    MotorActPos : DINT ;
    SwsMin : DINT ;
    SwsMax : DINT ;
    PresetPos : DINT ;
    PresetData : DINT ;
    AreaWin : DINT ;
    PosWin : DINT ;
    Encoder : DINT ;
    _09 : DINT ;
    _10 : DINT ;
    _11 : DINT ;
    _12 : DINT ;
    _13 : DINT ;
    _14 : DINT ;
    _15 : DINT ;
    _16 : DINT ;
    _17 : DINT ;
    _18 : DINT ;
    Offset : DINT ;
    ManPrevPos : DINT ;
    ManActPos : DINT ;
    ManNextPos : DINT ;
    ManMinPos : DINT ;
    ManMaxPos : DINT ;
    ManTargPosVal : DINT ;
    _26 : DINT ;
    _27 : DINT ;
    _28 : DINT ;
    _29 : DINT ;
    _30 : DINT ;
    _31 : DINT ;
    _32 : DINT ;
    _33 : DINT ;
    _34 : DINT ;
    ActPosMinusOffset : DINT ;
    TargPosPlusOffset : DINT ;
    _37 : DINT ;
    _38 : DINT ;
    _39 : DINT ;
    _40 : DINT ;
    _41 : DINT ;
    _42 : DINT ;
    _43 : DINT ;
    _44 : DINT ;
    _45 : DINT ;
    _46 : DINT ;
    _47 : DINT ;
    _48 : DINT ;
    _49 : DINT ;
    _50 : DINT ;
    _51 : DINT ;
    _52 : DINT ;
    _53 : DINT ;
    _54 : DINT ;
    _55 : DINT ;
    _56 : DINT ;
    _57 : DINT ;
    _58 : DINT ;
    _59 : DINT ;
    _60 : DINT ;
    _61 : DINT ;
    _62 : DINT ;
    _63 : DINT ;
    _64 : DINT ;
    _65 : DINT ;
    _66 : DINT ;
    _67 : DINT ;
    _68 : DINT ;
    _69 : DINT ;
    _70 : DINT ;
    _71 : DINT ;
    _72 : DINT ;
    _73 : DINT ;
    _74 : DINT ;
   END_STRUCT ;
   _i : STRUCT
    MotorIn_00 : INT ;
    MotorIn_01 : INT ;
    MotorIn_02 : INT ;
    MotorIn_03 : INT ;
    MotorIn_04 : INT ;
    MotorIn_05 : INT ;
    MotorOut_00 : INT ;
    MotorOut_01 : INT ;
    MotorOut_02 : INT ;
    MotorOut_03 : INT ;
    MotorOut_04 : INT ;
    MotorOut_05 : INT ;
    MotorCrtWord : INT ;
    MotorTargSpeed : INT ;
    MotorTargAcc : INT ;
    MotorTargDeacc : INT ;
    MotorStateWord : INT ;
    MotorActSpeed : INT ;
    MotorActCurrent : INT ;
    MotorActWorkLoad : INT ;
    SourcePosNo : INT ;
    TargPosNo : INT ;
    ActAreaNo : INT ;
    ServiceV : INT ;
    ManualV : INT ;
    OnlineV : INT ;
    ForcedSlowV : INT ;
    RuntimeSec : INT ;
    ActPosNo : INT ;
    ScanAreaNo : INT ;
    SpeedManual : INT ;
    SafetySpeed : INT ;	//sichere Geschwindigkeit (1/min)
    SpeedForcSlow : INT ;
    SpeedManSlo : INT ;
    Acceleration : INT ;
    Deacceleration : INT ;
    _36 : INT ;
    ManTargPosNo : INT ;
    PrevPosNo : INT ;
    NextPosNo : INT ;
    MinPosNo : INT ;
    MaxPosNo : INT ;
    _42 : INT ;
    _43 : INT ;
    _44 : INT ;
    ActLIF_DBNo : INT ;
    _46 : INT ;
    _47 : INT ;
    _48 : INT ;
    _49 : INT ;
    _50 : INT ;
    _51 : INT ;
    _52 : INT ;
    _53 : INT ;
    _54 : INT ;
    _55 : INT ;
    _56 : INT ;
    _57 : INT ;
    _58 : INT ;
    _59 : INT ;
    _60 : INT ;
    _61 : INT ;
    _62 : INT ;
    _63 : INT ;
    _64 : INT ;
    _65 : INT ;
    _66 : INT ;
    _67 : INT ;
    _68 : INT ;
    _69 : INT ;
    _70 : INT ;
    _71 : INT ;
    _72 : INT ;
    _73 : INT ;
    _74 : INT ;
    _75 : INT ;
    _76 : INT ;
    _77 : INT ;
    _78 : INT ;
    _79 : INT ;
    _80 : INT ;
    _81 : INT ;
    _82 : INT ;
    _83 : INT ;
    _84 : INT ;
    _85 : INT ;
    _86 : INT ;
    _87 : INT ;
    _88 : INT ;
    _89 : INT ;
    _90 : INT ;
    _91 : INT ;
    _92 : INT ;
    _93 : INT ;
    _94 : INT ;
    _95 : INT ;
    _96 : INT ;
    _97 : INT ;
    _98 : INT ;
    DriveErrorCode : INT ;
   END_STRUCT ;
   _x : STRUCT
    InchMinus : BOOL ;
    InchPlus : BOOL ;
    TargIsPos : BOOL ;
    RelForPos : BOOL ;
    MovesMinus : BOOL ;
    MovesPlus : BOOL ;
    Moves : BOOL ;
    InArea : BOOL ;
    InPos : BOOL ;
    FastStop : BOOL ;
    ManPosFound : BOOL ;
    MotorReady : BOOL ;
    MotorRefOk : BOOL ;
    ForcedSlow : BOOL ;
    StartPos : BOOL ;
    Position_Found : BOOL ;
    pFl_StartPos : BOOL ;
    _17 : BOOL ;
    DelayFaststop : BOOL ;
    ReleaseScan : BOOL ;
    ScanInPos : BOOL ;
    AutoInPos : BOOL ;
    TargPosFront : BOOL ;
    TargPosBack : BOOL ;
    InPosCart : BOOL ;
    _25 : BOOL ;
    _26 : BOOL ;
    _27 : BOOL ;
    _28 : BOOL ;
    _29 : BOOL ;
    _30 : BOOL ;
    _31 : BOOL ;
    _32 : BOOL ;
    _33 : BOOL ;
    _34 : BOOL ;
    _35 : BOOL ;
    _36 : BOOL ;
    _37 : BOOL ;
    _38 : BOOL ;
    _39 : BOOL ;
    _40 : BOOL ;
    _41 : BOOL ;
    _42 : BOOL ;
    _43 : BOOL ;
    _44 : BOOL ;
    _45 : BOOL ;
    _46 : BOOL ;
    _47 : BOOL ;
    _48 : BOOL ;
    _49 : BOOL ;
    _50 : BOOL ;
    PresetOffset : BOOL ;
    _52 : BOOL ;
    _53 : BOOL ;
    _54 : BOOL ;
    _55 : BOOL ;
    _56 : BOOL ;
    _57 : BOOL ;
    _58 : BOOL ;
    _59 : BOOL ;
    _60 : BOOL ;
    _61 : BOOL ;
    fs_Minus_SW : BOOL ;	//forced slow software
    fs_Plus_Sw : BOOL ;	//forced slow software
    _64 : BOOL ;
    _65 : BOOL ;
    _66 : BOOL ;
    _67 : BOOL ;
    _68 : BOOL ;
    _69 : BOOL ;
    _70 : BOOL ;
    _71 : BOOL ;
    _72 : BOOL ;
    _73 : BOOL ;
    _74 : BOOL ;
    _75 : BOOL ;
    _76 : BOOL ;
    _77 : BOOL ;
    _78 : BOOL ;
    _79 : BOOL ;
    _80 : BOOL ;
    _81 : BOOL ;
    _82 : BOOL ;
    _83 : BOOL ;
    _84 : BOOL ;
    _85 : BOOL ;
    _86 : BOOL ;
    _87 : BOOL ;
    _88 : BOOL ;
    _89 : BOOL ;
    _90 : BOOL ;
    _91 : BOOL ;
    _92 : BOOL ;
    _93 : BOOL ;
    _94 : BOOL ;
    _95 : BOOL ;
   END_STRUCT ;
  END_STRUCT ;	
BEGIN
   _di.MotorTargPos := L#33953;
   _di.MotorActPos := L#33953;
   _di.SwsMin := L#6900;
   _di.SwsMax := L#37060;
   _di.AreaWin := L#10;
   _di.PosWin := L#1;
   _di.Encoder := L#33946;
   _di.ManPrevPos := L#5134;
   _di.ManActPos := L#7046;
   _di.ManNextPos := L#9344;
   _di.ManMinPos := L#1313;
   _di.ManMaxPos := L#9344;
   _di.ManTargPosVal := L#3223;
   _di.ActPosMinusOffset := L#33953;
   _di.TargPosPlusOffset := L#33953;
   _i.MotorIn_00 := 526;
   _i.MotorIn_02 := -31583;
   _i.MotorIn_05 := 140;
   _i.MotorOut_00 := 6144;
   _i.MotorOut_02 := -31583;
   _i.MotorOut_03 := 1160;
   _i.MotorOut_04 := 2600;
   _i.MotorOut_05 := 2600;
   _i.MotorCrtWord := 6144;
   _i.MotorTargSpeed := 1160;
   _i.MotorTargAcc := 2600;
   _i.MotorTargDeacc := 2600;
   _i.MotorStateWord := 526;
   _i.MotorActWorkLoad := 140;
   _i.TargPosNo := 2;
   _i.ActAreaNo := 4;
   _i.ServiceV := 1;
   _i.ManualV := 30;
   _i.OnlineV := 100;
   _i.ForcedSlowV := 5;
   _i.ActPosNo := 2;
   _i.ScanAreaNo := 2;
   _i.SpeedManual := 2;
   _i.SpeedForcSlow := 5;
   _i.SpeedManSlo := 2;
   _i.Acceleration := 3000;
   _i.Deacceleration := 3000;
   _i._36 := 2;
   _i.ManTargPosNo := 2;
   _i.PrevPosNo := 3;
   _i.NextPosNo := 5;
   _i.MinPosNo := 1;
   _i.MaxPosNo := 5;
   _i.ActLIF_DBNo := 201;
   _i.DriveErrorCode := 2;
   _x.InArea := TRUE;
   _x.FastStop := TRUE;
   _x.MotorReady := TRUE;
   _x.MotorRefOk := TRUE;
   _x.Position_Found := TRUE;
   _x.ScanInPos := TRUE;
   _x.AutoInPos := TRUE;
END_DATA_BLOCK

DATA_BLOCK "DB_ComGateway"	// DB 10
VERSION : 0.1
  STRUCT
   TM : STRUCT
    StateWord : INT ;
    TotalLength : INT ;
    FaceLength : INT ;
    Circum : INT ;
    BriActPos : INT ;
    TroActPos : INT ;
    LifActPos : INT ;
    TelActPos : INT ;
    WidActPos : INT ;
    Ax05ActPos : INT ;
    Ax06ActPos : INT ;
    Ax07ActPos : INT ;
    Ax08ActPos : INT ;
    Ax09ActPos : INT ;
    BriMotorPos : DINT ;
    TroMotorPos : DINT ;
    LifMotorPos : DINT ;
    TelMotorPos : DINT ;
    WidMotorPos : DINT ;
    Ax05MotorPos : DINT ;
    Ax06MotorPos : DINT ;
    Ax07MotorPos : DINT ;
    Ax08MotorPos : DINT ;
    Ax09MotorPos : DINT ;
    ParaCnt : INT ;
    ParaNo : INT ;
    ParaData : DINT ;
    Err00 : INT ;
    Err01 : INT ;
    Err02 : INT ;
    Err03 : INT ;
    Err04 : INT ;
    Err05 : INT ;
    Err06 : INT ;
    Err07 : INT ;
    Err08 : INT ;
    Err09 : INT ;
    Err10 : INT ;
    Err11 : INT ;
    StepNo : INT ;
    WorkHours : DINT ;
    _53 : INT ;
    _54 : INT ;
    CommCounterToMaster : INT ;
    _56 : INT ;
    _57 : INT ;
    _58 : INT ;
    InvStateWord : INT ;
    Lifebit : BOOL ;
    TeleskopsFree : BOOL ;
    Buffer_Free : BOOL ;
    LiftTop : BOOL ;
    Online : BOOL ;
    ReadyOnline : BOOL ;
    Error : BOOL ;
    MovingSource : BOOL ;
    MovingTarget : BOOL ;
    TeleskopCenterpos : BOOL ;
    OrderRunning : BOOL ;
    OrderEnd : BOOL ;
    OrderPaused : BOOL ;
    Bit13 : BOOL ;
    TargetNok : BOOL ;
    RequestTurne : BOOL ;
    Spare122 : WORD ;
    Spare124 : WORD ;
    Spare126 : WORD ;
    Move : UDT 7;
    Spare154 : WORD ;
    Spare156 : WORD ;
    Spare158 : WORD ;
    ErrorCabinet : STRUCT
     Err00 : INT ;
     Err01 : INT ;
     Err02 : INT ;
     Err03 : INT ;
     Err04 : INT ;
     Err05 : INT ;
     Err06 : INT ;
     Err07 : INT ;
     Err08 : INT ;
     Err09 : INT ;
     Err10 : INT ;
     Err11 : INT ;
    END_STRUCT ;
    LS_1 : STRUCT
     SPARE_00 : BOOL ;
     SPARE_01 : BOOL ;
     SPARE_02 : BOOL ;
     SPARE_03 : BOOL ;
     SPARE_04 : BOOL ;
     SPARE_05 : BOOL ;
     Online : BOOL ;
     Ready : BOOL ;
     Palette_In_Station : BOOL ;
     Pos_11_Free : BOOL ;
     Pos_12_Free : BOOL ;
     SPARE_13 : BOOL ;
     SPARE_14 : BOOL ;
     SPARE_15 : BOOL ;
     SPARE_16 : BOOL ;
     SPARE_17 : BOOL ;
    END_STRUCT ;
    LS_2 : STRUCT
     SPARE_00 : BOOL ;
     SPARE_01 : BOOL ;
     SPARE_02 : BOOL ;
     SPARE_03 : BOOL ;
     SPARE_04 : BOOL ;
     SPARE_05 : BOOL ;
     Online : BOOL ;
     Ready : BOOL ;
     Palette_In_Station : BOOL ;
     Pos_11_Free : BOOL ;
     Pos_12_Free : BOOL ;
     SPARE_13 : BOOL ;
     SPARE_14 : BOOL ;
     SPARE_15 : BOOL ;
     SPARE_16 : BOOL ;
     SPARE_17 : BOOL ;
    END_STRUCT ;
    LS_3 : STRUCT
     SPARE_00 : BOOL ;
     SPARE_01 : BOOL ;
     SPARE_02 : BOOL ;
     SPARE_03 : BOOL ;
     SPARE_04 : BOOL ;
     SPARE_05 : BOOL ;
     Online : BOOL ;
     Ready : BOOL ;
     Palette_In_Station : BOOL ;
     Pos_11_Free : BOOL ;
     Pos_12_Free : BOOL ;
     SPARE_13 : BOOL ;
     SPARE_14 : BOOL ;
     SPARE_15 : BOOL ;
     SPARE_16 : BOOL ;
     SPARE_17 : BOOL ;
    END_STRUCT ;
    Spare : ARRAY  [1 .. 5 ] OF WORD ;
   END_STRUCT ;
   FM : STRUCT
    ReleaseManual : BOOL ;
    spare01 : BOOL ;
    StartOrder : BOOL ;
    CleareOrder : BOOL ;
    StopOrder : BOOL ;
    spare05 : BOOL ;
    spare06 : BOOL ;
    ReleaseOnline : BOOL ;
    Lifebit : BOOL ;
    spare11 : BOOL ;
    StartBasePos : BOOL ;
    ChangeOrder : BOOL ;
    QuitOrderFinished : BOOL ;
    ResetErrors : BOOL ;
    ServiceOn : BOOL ;
    BypassLimmitsOn : BOOL ;
    TotalLength : INT ;
    FaceLength : INT ;
    Circum : INT ;
    SourceBri : INT ;
    SourceTro : INT ;
    SourceLif : INT ;
    SourceTel : INT ;
    SourceAx04 : INT ;
    SourceAx05 : INT ;
    SourceAx06 : INT ;
    SourceAx07 : INT ;
    SourceAx08 : INT ;
    SourceAx09 : INT ;
    TargBri : INT ;
    TargTro : INT ;
    TargLif : INT ;
    TargTel : INT ;
    TargAx04 : INT ;
    TargAx05 : INT ;
    TargAx06 : INT ;
    TargAx07 : INT ;
    TargAx08 : INT ;
    TargAx09 : INT ;
    Occ00 : INT ;
    Occ01 : INT ;
    Occ02 : INT ;
    Occ03 : INT ;
    SafetyAreas00 : INT ;
    SafetyAreas01 : INT ;
    ParaCnt : INT ;
    ParaNo : INT ;
    ParaData : DINT ;
    _34 : INT ;
    _35 : INT ;
    _36 : INT ;
    _37 : INT ;
    _38 : INT ;
    _39 : INT ;
    _40 : INT ;
    _41 : INT ;
    _42 : INT ;
    _43 : INT ;
    _44 : INT ;
    CommCounterFromMaster : INT ;
    _46 : INT ;
    _47 : INT ;
    _48 : INT ;
    InvCrtWord : INT ;
    Bit100_0 : BOOL ;
    Bit100_1 : BOOL ;
    Bit100_2 : BOOL ;
    Bit100_3 : BOOL ;
    Bit100_4 : BOOL ;
    Bit100_5 : BOOL ;
    Bit00_6 : BOOL ;
    Bit100_7 : BOOL ;
    Release : BOOL ;
    BypassLimits : BOOL ;
    Service : BOOL ;
    Sw_Manual : BOOL ;
    Bit101_4 : BOOL ;
    Bit101_5 : BOOL ;
    Bit101_6 : BOOL ;
    Bit101_7 : BOOL ;
    BrPosRelease : INT ;
    TrPosRelease : INT ;
    LiPosRelease : INT ;
    TlPosRelease : INT ;
    spare_110 : INT ;
    spare_112 : INT ;
    spare_114 : INT ;
    spare_116 : INT ;
    spare_118 : INT ;
    spare_120 : INT ;
    spare_122 : INT ;
    spare_124 : INT ;
    spare_126 : INT ;
    Move : UDT 7;
    LS_1 : STRUCT
     Start_Load : BOOL ;
     Start_Unload : BOOL ;
     Step_Load : BOOL ;
     Step_Unload : BOOL ;
     CleareOrder : BOOL ;
     SPARE_05 : BOOL ;
     SPARE_06 : BOOL ;
     SPARE_07 : BOOL ;
     SPARE_10 : BOOL ;
     SPARE_11 : BOOL ;
     SPARE_12 : BOOL ;
     SPARE_13 : BOOL ;
     SPARE_14 : BOOL ;
     SPARE_15 : BOOL ;
     SPARE_16 : BOOL ;
     SPARE_17 : BOOL ;
     TotalLength : INT ;
     FaceLength : INT ;
     Circum : INT ;
    END_STRUCT ;
    Spare : ARRAY  [1 .. 19 ] OF WORD ;
   END_STRUCT ;
  END_STRUCT ;	
BEGIN
   TM.StateWord := 48;
   TM.BriActPos := 2;
   TM.TroActPos := 1;
   TM.Ax07ActPos := 1;
   TM.BriMotorPos := L#33953;
   TM.CommCounterToMaster := 9772;
   TM.Online := TRUE;
   TM.ReadyOnline := TRUE;
   TM.Move.Action := 3;
   TM.Move.Value_01 := 2;
   TM.Move.Value_02 := 1;
   TM.Move.Value_08 := 1;
   TM.LS_1.Online := TRUE;
   TM.LS_1.Ready := TRUE;
   TM.LS_1.Palette_In_Station := TRUE;
   TM.LS_1.Pos_11_Free := TRUE;
   TM.LS_1.Pos_12_Free := TRUE;
   TM.LS_2.Online := TRUE;
   TM.LS_2.Ready := TRUE;
   TM.LS_2.Palette_In_Station := TRUE;
   TM.LS_2.Pos_11_Free := TRUE;
   TM.LS_2.Pos_12_Free := TRUE;
   TM.LS_3.Online := TRUE;
   TM.LS_3.Ready := TRUE;
   TM.LS_3.Palette_In_Station := TRUE;
   TM.LS_3.Pos_11_Free := TRUE;
   TM.LS_3.Pos_12_Free := TRUE;
   TM.Spare[1] := W#16#4241;
   TM.Spare[2] := W#16#5545;
   TM.Spare[3] := W#16#5520;
   FM.TargBri := 2;
   FM.TargTro := 1;
   FM.TargLif := 100;
   FM.TargTel := 100;
   FM.TargAx04 := 8480;
   FM.ParaCnt := 321;
   FM.ParaNo := 654;
   FM.ParaData := L#76542;
   FM.CommCounterFromMaster := 9771;
   FM.Bit100_1 := TRUE;
   FM.Bit100_2 := TRUE;
   FM.Move.MsgCounter := 682;
   FM.Move.Action := 3;
   FM.Move.Value_01 := 2;
   FM.Move.Value_02 := 1;
END_DATA_BLOCK

DATA_BLOCK "IDB_FB2_BRI"	// DB 11
AUTHOR : Koenig
VERSION : 0.0
"MovidriveB_Control"
BEGIN
END_DATA_BLOCK

DATA_BLOCK "DB_OrderBuffer"	// DB 15
VERSION : 0.1
  STRUCT
   SourceBri : INT ;
   SourceTro : INT ;
   SourceLif : INT ;
   SourceTel : INT ;
   TargetBri : INT ;
   TargetTro : INT ;
   TargetLif : INT ;
   TargetTel : INT ;
   OrderTotalLength : INT ;
   OrderFaceLength : INT ;
   OrderCircum : INT ;
  END_STRUCT ;	
BEGIN
   TargetBri := 2;
   TargetTro := 1;
   TargetLif := 100;
   TargetTel := 100;
END_DATA_BLOCK

DATA_BLOCK "DB_TargetData"	// DB 19
VERSION : 0.1
  STRUCT
   BrPosNo : INT  := 1;
   BrPosVal : DINT  := L#1000;
   TrPosNo : INT  := 1;
   TrPosVal : DINT ;
   LiPosNo : INT ;
   LiPosValHo : DINT ;
   LiPosValHu : DINT ;
   TlPosNo : INT ;
   TlPosVal : DINT ;
   Hooktype : INT ;
   CircumMax : INT ;
   Reserve : INT ;
   Hookdata : UDT 102;
  END_STRUCT ;	
BEGIN
   BrPosNo := 2;
   BrPosVal := L#33953;
   TrPosNo := 1;
END_DATA_BLOCK

DATA_BLOCK "IDB_MasterInterface"	// DB 33
VERSION : 0.0
"MasterInterface"
BEGIN
END_DATA_BLOCK

DATA_BLOCK "IDB_WREC_BR"	// DB 50
AUTHOR : SIMATIC
FAMILY : DP
VERSION : 0.0
"WRREC"
BEGIN
END_DATA_BLOCK

DATA_BLOCK "INOUT"	// DB 80
VERSION : 0.1
  STRUCT
   IN : STRUCT
    CAB_PhaseOK : BOOL ;
    CAB_24V_OK : BOOL ;
    CAB_115V_OK : BOOL ;
    CAB_400V_OK : BOOL ;
    CAB_SW_Preset_BRI : BOOL ;
    CAB_HighTemp : BOOL ;
    CAB_TS_Reset : BOOL ;
    CAB_Power_Brakes_OK : BOOL ;
    CAB_Power_Fan : BOOL ;
    CAB_Temp_Warning : BOOL ;
    Spare_01 : WORD ;
    Spare_02 : WORD ;
    BRI_ForcedSlow_plus_NO : BOOL ;
    BRI_ForcedSlow_plus_NC : BOOL ;
    BRI_ForcedSlow_minus_NO : BOOL ;
    BRI_ForcedSlow_minus_NC : BOOL ;
    BRI_Limit_plus : BOOL ;
    BRI_Limit_minus : BOOL ;
    RC_BRI_Plus : BOOL ;
    RC_BRI_Minus : BOOL ;
    RC_BRI_FastPlus : BOOL ;
    RC_BRI_FastMinus : BOOL ;
    Spare_03 : WORD ;
    Spare_04 : WORD ;
    TRO_isOnCarrier : BOOL ;
   END_STRUCT ;
   Spare : ARRAY  [1 .. 18 ] OF WORD ;
   OUT : STRUCT
    CAB_Horn : BOOL ;
    CAB_LP_State_0 : BOOL ;
    CAB_LP_State_1 : BOOL ;
    CAB_LP_State_2 : BOOL ;
    CAB_LP_Reset : BOOL ;
    CAB_LP_Preset : BOOL ;
    CAB_Reset_24V : BOOL ;
    CAB_Reset_EOFF : BOOL ;
   END_STRUCT ;
  END_STRUCT ;	
BEGIN
   IN.CAB_PhaseOK := TRUE;
   IN.CAB_24V_OK := TRUE;
   IN.CAB_115V_OK := TRUE;
   IN.CAB_400V_OK := TRUE;
   IN.CAB_Power_Brakes_OK := TRUE;
   IN.CAB_Power_Fan := TRUE;
   IN.BRI_ForcedSlow_plus_NC := TRUE;
   IN.BRI_ForcedSlow_minus_NC := TRUE;
   OUT.CAB_LP_State_1 := TRUE;
END_DATA_BLOCK

DATA_BLOCK "Moves"	// DB 101
VERSION : 0.1
  STRUCT
   PC : UDT 7;
   Unit : ARRAY  [1 .. 50 ] OF UDT 7;
  END_STRUCT ;	
BEGIN
   PC.MsgCounter := 682;
   PC.Action := 3;
   PC.Value_01 := 2;
   PC.Value_02 := 1;
   Unit[1].Action := 3;
   Unit[1].Value_01 := 2;
   Unit[1].Value_02 := 1;
   Unit[1].Value_08 := 1;
END_DATA_BLOCK

DATA_BLOCK "InstanzDB PNIODiag"	// DB 126
AUTHOR : ICom
FAMILY : DIAGNOSE
VERSION : 0.0
"PNIODiag"
BEGIN
END_DATA_BLOCK

DATA_BLOCK "InstanzDB STATDiag"	// DB 127
AUTHOR : ICom
FAMILY : DIAGNOSE
VERSION : 0.0
"STATDiag"
BEGIN
END_DATA_BLOCK

DATA_BLOCK "DB_Steps"	// DB 132
VERSION : 0.1
  STRUCT
   _DINT : STRUCT
    StepsStartet : DINT ;
    StepsFinished : DINT ;
    _02 : DINT ;
    _03 : DINT ;
    _04 : DINT ;
    _05 : DINT ;
    _06 : DINT ;
    _07 : DINT ;
    _08 : DINT ;
    _09 : DINT ;
    _10 : DINT ;
    _11 : DINT ;
    _12 : DINT ;
    _13 : DINT ;
    _14 : DINT ;
    _15 : DINT ;
    _16 : DINT ;
    _17 : DINT ;
    _18 : DINT ;
    _19 : DINT ;
    _20 : DINT ;
    _21 : DINT ;
    _22 : DINT ;
    _23 : DINT ;
    _24 : DINT ;
    _25 : DINT ;
    _26 : DINT ;
    _27 : DINT ;
    _28 : DINT ;
    _29 : DINT ;
    _30 : DINT ;
    _31 : DINT ;
    _32 : DINT ;
    _33 : DINT ;
    _34 : DINT ;
    _35 : DINT ;
    _36 : DINT ;
    _37 : DINT ;
    _38 : DINT ;
    _39 : DINT ;
    _40 : DINT ;
    _41 : DINT ;
    _42 : DINT ;
    _43 : DINT ;
    _44 : DINT ;
    _45 : DINT ;
    _46 : DINT ;
    _47 : DINT ;
    _48 : DINT ;
    _49 : DINT ;
    _50 : DINT ;
    _51 : DINT ;
    _52 : DINT ;
    _53 : DINT ;
    _54 : DINT ;
    _55 : DINT ;
    _56 : DINT ;
    _57 : DINT ;
    _58 : DINT ;
    _59 : DINT ;
    _60 : DINT ;
    _61 : DINT ;
    _62 : DINT ;
    _63 : DINT ;
    _64 : DINT ;
    _65 : DINT ;
    _66 : DINT ;
    _67 : DINT ;
    _68 : DINT ;
    _69 : DINT ;
    _70 : DINT ;
    _71 : DINT ;
    _72 : DINT ;
    _73 : DINT ;
    _74 : DINT ;
    _75 : DINT ;
    _76 : DINT ;
    _77 : DINT ;
    _78 : DINT ;
    _79 : DINT ;
    _80 : DINT ;
    _81 : DINT ;
    _82 : DINT ;
    _83 : DINT ;
    _84 : DINT ;
    _85 : DINT ;
    _86 : DINT ;
    _87 : DINT ;
    _88 : DINT ;
    _89 : DINT ;
    _90 : DINT ;
    _91 : DINT ;
    _92 : DINT ;
    _93 : DINT ;
    _94 : DINT ;
    _95 : DINT ;
    _96 : DINT ;
    _97 : DINT ;
    _98 : DINT ;
    _99 : DINT ;
    _100 : DINT ;
    _101 : DINT ;
    _102 : DINT ;
    _103 : DINT ;
    _104 : DINT ;
    _105 : DINT ;
    _106 : DINT ;
    _107 : DINT ;
    _108 : DINT ;
    _109 : DINT ;
    _110 : DINT ;
    _111 : DINT ;
    _112 : DINT ;
    _113 : DINT ;
    _114 : DINT ;
    _115 : DINT ;
    _116 : DINT ;
    _117 : DINT ;
    _118 : DINT ;
    _119 : DINT ;
    _120 : DINT ;
    _121 : DINT ;
    _122 : DINT ;
    _123 : DINT ;
    _124 : DINT ;
    _125 : DINT ;
    _126 : DINT ;
    _127 : DINT ;
    _128 : DINT ;
    _129 : DINT ;
    _130 : DINT ;
    _131 : DINT ;
    _132 : DINT ;
    _133 : DINT ;
    _134 : DINT ;
    _135 : DINT ;
    _136 : DINT ;
    _137 : DINT ;
    _138 : DINT ;
    _139 : DINT ;
    _140 : DINT ;
    _141 : DINT ;
    _142 : DINT ;
    _143 : DINT ;
    _144 : DINT ;
    _145 : DINT ;
    _146 : DINT ;
    _147 : DINT ;
    _148 : DINT ;
    _149 : DINT ;
    _150 : DINT ;
    _151 : DINT ;
    _152 : DINT ;
    _153 : DINT ;
    _154 : DINT ;
    _155 : DINT ;
    _156 : DINT ;
    _157 : DINT ;
    _158 : DINT ;
    _159 : DINT ;
   END_STRUCT ;
   _INT : STRUCT
    BASEPOS_Steps : INT ;
    EMPTY_Steps : INT ;
    GET_Steps : INT ;
    PUT_Steps : INT ;
    _04 : INT ;
    _05 : INT ;
    _06 : INT ;
    _07 : INT ;
    _08 : INT ;
    _09 : INT ;
    ChkHookOccCntGET : INT ;	//Check occupation sensors hook
    ChkHookOccCntPUT : INT ;
    _12 : INT ;
    _13 : INT ;
    _14 : INT ;
    _15 : INT ;
    _16 : INT ;
    _17 : INT ;
    _18 : INT ;
    _19 : INT ;
    _20 : INT ;
    _21 : INT ;
    _22 : INT ;
    _23 : INT ;
    _24 : INT ;
    _25 : INT ;
    _26 : INT ;
    _27 : INT ;
    _28 : INT ;
    _29 : INT ;
    _30 : INT ;
    _31 : INT ;
    _32 : INT ;
    _33 : INT ;
    _34 : INT ;
    _35 : INT ;
    _36 : INT ;
    _37 : INT ;
    _38 : INT ;
    _39 : INT ;
    _40 : INT ;
    _41 : INT ;
    _42 : INT ;
    _43 : INT ;
    _44 : INT ;
    _45 : INT ;
    _46 : INT ;
    _47 : INT ;
    _48 : INT ;
    _49 : INT ;
    _50 : INT ;
    _51 : INT ;
    _52 : INT ;
    _53 : INT ;
    _54 : INT ;
    _55 : INT ;
    _56 : INT ;
    _57 : INT ;
    _58 : INT ;
    _59 : INT ;
    _60 : INT ;
    _61 : INT ;
    _62 : INT ;
    _63 : INT ;
    _64 : INT ;
    _65 : INT ;
    _66 : INT ;
    _67 : INT ;
    _68 : INT ;
    _69 : INT ;
    _70 : INT ;
    _71 : INT ;
    _72 : INT ;
    _73 : INT ;
    _74 : INT ;
    _75 : INT ;
    _76 : INT ;
    _77 : INT ;
    _78 : INT ;
    _79 : INT ;
    _80 : INT ;
    _81 : INT ;
    _82 : INT ;
    _83 : INT ;
    _84 : INT ;
    _85 : INT ;
    _86 : INT ;
    _87 : INT ;
    _88 : INT ;
    _89 : INT ;
    _90 : INT ;
    _91 : INT ;
    _92 : INT ;
    _93 : INT ;
    _94 : INT ;
    _95 : INT ;
    _96 : INT ;
    _97 : INT ;
    _98 : INT ;
    _99 : INT ;
    _100 : INT ;
    _101 : INT ;
    _102 : INT ;
    _103 : INT ;
    _104 : INT ;
    _105 : INT ;
    _106 : INT ;
    _107 : INT ;
    _108 : INT ;
    _109 : INT ;
    _110 : INT ;
    _111 : INT ;
    _112 : INT ;
    _113 : INT ;
    _114 : INT ;
    _115 : INT ;
    _116 : INT ;
    _117 : INT ;
    _118 : INT ;
    _119 : INT ;
    _120 : INT ;
    _121 : INT ;
    _122 : INT ;
    _123 : INT ;
    _124 : INT ;
    _125 : INT ;
    _126 : INT ;
    _127 : INT ;
    _128 : INT ;
    _129 : INT ;
    _130 : INT ;
    _131 : INT ;
    _132 : INT ;
    _133 : INT ;
    _134 : INT ;
    _135 : INT ;
    _136 : INT ;
    _137 : INT ;
    _138 : INT ;
    _139 : INT ;
    _140 : INT ;
    _141 : INT ;
    _142 : INT ;
    _143 : INT ;
    _144 : INT ;
    _145 : INT ;
    _146 : INT ;
    _147 : INT ;
    _148 : INT ;
    _149 : INT ;
    _150 : INT ;
    _151 : INT ;
    _152 : INT ;
    _153 : INT ;
    _154 : INT ;
    _155 : INT ;
    _156 : INT ;
    _157 : INT ;
    _158 : INT ;
    _159 : INT ;
   END_STRUCT ;
   _BOOL : STRUCT
    Target_DataOK : BOOL ;
    _01 : BOOL ;
    _02 : BOOL ;
    _03 : BOOL ;
    _04 : BOOL ;
    _05 : BOOL ;
    _06 : BOOL ;
    _07 : BOOL ;
    BASEPOS_Req : BOOL ;
    EMPTY_Req : BOOL ;
    GET_Req : BOOL ;
    PUT_Req : BOOL ;
    BASEPOS_active : BOOL ;
    EMPTY_active : BOOL ;
    GET_active : BOOL ;
    PUT_active : BOOL ;
    STEPS_active : BOOL ;
    STEPS_start : BOOL ;
    GET_Finished : BOOL ;
    _19 : BOOL ;
    _20 : BOOL ;
    _21 : BOOL ;
    _22 : BOOL ;
    _23 : BOOL ;
    _24 : BOOL ;
    _25 : BOOL ;
    _26 : BOOL ;
    _27 : BOOL ;
    _28 : BOOL ;
    _29 : BOOL ;
    _30 : BOOL ;
    _31 : BOOL ;
    ChkHookOccGET : BOOL ;
    ChkHookOccGET_End : BOOL ;
    ChkHookOccGET_OK : BOOL ;
    ChkHookOccPUT : BOOL ;
    ChkHookOccPUT_End : BOOL ;
    ChkHookOccPUT_OK : BOOL ;
    ChkHookOcxGET_enable : BOOL ;
    ChkHookOcxPUT_enable : BOOL ;
    _40 : BOOL ;
    _41 : BOOL ;
    _42 : BOOL ;
    _43 : BOOL ;
    _44 : BOOL ;
    _45 : BOOL ;
    _46 : BOOL ;
    _47 : BOOL ;
    _48 : BOOL ;
    _49 : BOOL ;
    _50 : BOOL ;
    _51 : BOOL ;
    _52 : BOOL ;
    _53 : BOOL ;
    _54 : BOOL ;
    _55 : BOOL ;
    _56 : BOOL ;
    _57 : BOOL ;
    _58 : BOOL ;
    _59 : BOOL ;
    _60 : BOOL ;
    _61 : BOOL ;
    _62 : BOOL ;
    _63 : BOOL ;
    _64 : BOOL ;
    _65 : BOOL ;
    _66 : BOOL ;
    _67 : BOOL ;
    _68 : BOOL ;
    _69 : BOOL ;
    _70 : BOOL ;
    _71 : BOOL ;
    _72 : BOOL ;
    _73 : BOOL ;
    _74 : BOOL ;
    _75 : BOOL ;
    _76 : BOOL ;
    _77 : BOOL ;
    _78 : BOOL ;
    _79 : BOOL ;
    _80 : BOOL ;
    _81 : BOOL ;
    _82 : BOOL ;
    _83 : BOOL ;
    _84 : BOOL ;
    _85 : BOOL ;
    _86 : BOOL ;
    _87 : BOOL ;
    _88 : BOOL ;
    _89 : BOOL ;
    _90 : BOOL ;
    _91 : BOOL ;
    _92 : BOOL ;
    _93 : BOOL ;
    _94 : BOOL ;
    _95 : BOOL ;
    _96 : BOOL ;
    _97 : BOOL ;
    _98 : BOOL ;
    _99 : BOOL ;
    _100 : BOOL ;
    _101 : BOOL ;
    _102 : BOOL ;
    _103 : BOOL ;
    _104 : BOOL ;
    _105 : BOOL ;
    _106 : BOOL ;
    _107 : BOOL ;
    _108 : BOOL ;
    _109 : BOOL ;
    _110 : BOOL ;
    _111 : BOOL ;
    _112 : BOOL ;
    _113 : BOOL ;
    _114 : BOOL ;
    _115 : BOOL ;
    _116 : BOOL ;
    _117 : BOOL ;
    _118 : BOOL ;
    _119 : BOOL ;
    _120 : BOOL ;
    _121 : BOOL ;
    _122 : BOOL ;
    _123 : BOOL ;
    _124 : BOOL ;
    _125 : BOOL ;
    _126 : BOOL ;
    _127 : BOOL ;
    _128 : BOOL ;
    _129 : BOOL ;
    _130 : BOOL ;
    _131 : BOOL ;
    _132 : BOOL ;
    _133 : BOOL ;
    _134 : BOOL ;
    _135 : BOOL ;
    _136 : BOOL ;
    _137 : BOOL ;
    _138 : BOOL ;
    _139 : BOOL ;
    _140 : BOOL ;
    _141 : BOOL ;
    _142 : BOOL ;
    _143 : BOOL ;
    _144 : BOOL ;
    _145 : BOOL ;
    _146 : BOOL ;
    _147 : BOOL ;
    _148 : BOOL ;
    _149 : BOOL ;
    _150 : BOOL ;
    _151 : BOOL ;
    _152 : BOOL ;
    _153 : BOOL ;
    _154 : BOOL ;
    _155 : BOOL ;
    _156 : BOOL ;
    _157 : BOOL ;
    _158 : BOOL ;
    _159 : BOOL ;
   END_STRUCT ;
  END_STRUCT ;	
BEGIN
   _DINT.StepsStartet := L#23778;
   _DINT.StepsFinished := L#376565;
   _INT.ChkHookOccCntGET := 5;
   _INT.ChkHookOccCntPUT := 3;
   _BOOL.ChkHookOcxGET_enable := TRUE;
   _BOOL.ChkHookOcxPUT_enable := TRUE;
END_DATA_BLOCK

DATA_BLOCK "COMM_CAR01"	// DB 150
AUTHOR : Koenig
VERSION : 0.1
  STRUCT
   TM : STRUCT
    StateWord : INT ;
    TotalLength : INT ;
    FaceLength : INT ;
    Circum : INT ;
    BriActPos : INT ;
    TroActPos : INT ;
    LifActPos : INT ;
    TelActPos : INT ;
    WidActPos : INT ;
    Ax05ActPos : INT ;
    Ax06ActPos : INT ;
    Ax07ActPos : INT ;
    Ax08ActPos : INT ;
    Ax09ActPos : INT ;
    BriMotorPos : DINT ;
    TroMotorPos : DINT ;
    LifMotorPos : DINT ;
    TelMotorPos : DINT ;
    WidMotorPos : DINT ;
    Ax05MotorPos : DINT ;
    Ax06MotorPos : DINT ;
    Ax07MotorPos : DINT ;
    Ax08MotorPos : DINT ;
    Ax09MotorPos : DINT ;
    ParaCnt : INT ;
    ParaNo : INT ;
    ParaData : DINT ;
    Err00 : INT ;
    Err01 : INT ;
    Err02 : INT ;
    Err03 : INT ;
    Err04 : INT ;
    Err05 : INT ;
    Err06 : INT ;
    Err07 : INT ;
    Err08 : INT ;
    Err09 : INT ;
    Err10 : INT ;
    Err11 : INT ;
    StepNo : INT ;
    WorkHours : DINT ;
    _53 : INT ;
    _54 : INT ;
    CommCounterToMaster : INT ;
    _56 : INT ;
    _57 : INT ;
    _58 : INT ;
    InvStateWord : INT ;
    Lifebit : BOOL ;
    TeleskopsFree : BOOL ;
    Buffer_Free : BOOL ;
    LiftTop : BOOL ;
    Online : BOOL ;
    ReadyOnline : BOOL ;
    Error : BOOL ;
    MovingSource : BOOL ;
    MovingTarget : BOOL ;
    TeleskopCenterpos : BOOL ;
    OrderRunning : BOOL ;
    OrderEnd : BOOL ;
    OrderPaused : BOOL ;
    Bit13 : BOOL ;
    TargetNok : BOOL ;
    RequestTurne : BOOL ;
    Spare122 : WORD ;
    Spare124 : WORD ;
    Spare126 : WORD ;
    Move : UDT 7;
    Spare154 : WORD ;
    Spare156 : WORD ;
    Spare158 : WORD ;
    ErrorCabinet : STRUCT
     Err00 : INT ;
     Err01 : INT ;
     Err02 : INT ;
     Err03 : INT ;
     Err04 : INT ;
     Err05 : INT ;
     Err06 : INT ;
     Err07 : INT ;
     Err08 : INT ;
     Err09 : INT ;
     Err10 : INT ;
     Err11 : INT ;
    END_STRUCT ;
    LS_1 : STRUCT
     SPARE_00 : BOOL ;
     SPARE_01 : BOOL ;
     SPARE_02 : BOOL ;
     SPARE_03 : BOOL ;
     SPARE_04 : BOOL ;
     SPARE_05 : BOOL ;
     Online : BOOL ;
     Ready : BOOL ;
     Palette_In_Station : BOOL ;
     Pos_11_Free : BOOL ;
     Pos_12_Free : BOOL ;
     SPARE_13 : BOOL ;
     SPARE_14 : BOOL ;
     SPARE_15 : BOOL ;
     SPARE_16 : BOOL ;
     SPARE_17 : BOOL ;
    END_STRUCT ;
    LS_2 : STRUCT
     SPARE_00 : BOOL ;
     SPARE_01 : BOOL ;
     SPARE_02 : BOOL ;
     SPARE_03 : BOOL ;
     SPARE_04 : BOOL ;
     SPARE_05 : BOOL ;
     Online : BOOL ;
     Ready : BOOL ;
     Palette_In_Station : BOOL ;
     Pos_11_Free : BOOL ;
     Pos_12_Free : BOOL ;
     SPARE_13 : BOOL ;
     SPARE_14 : BOOL ;
     SPARE_15 : BOOL ;
     SPARE_16 : BOOL ;
     SPARE_17 : BOOL ;
    END_STRUCT ;
    LS_3 : STRUCT
     SPARE_00 : BOOL ;
     SPARE_01 : BOOL ;
     SPARE_02 : BOOL ;
     SPARE_03 : BOOL ;
     SPARE_04 : BOOL ;
     SPARE_05 : BOOL ;
     Online : BOOL ;
     Ready : BOOL ;
     Palette_In_Station : BOOL ;
     Pos_11_Free : BOOL ;
     Pos_12_Free : BOOL ;
     SPARE_13 : BOOL ;
     SPARE_14 : BOOL ;
     SPARE_15 : BOOL ;
     SPARE_16 : BOOL ;
     SPARE_17 : BOOL ;
    END_STRUCT ;
    Spare : ARRAY  [1 .. 5 ] OF WORD ;
   END_STRUCT ;
   FM : STRUCT
    ReleaseManual : BOOL ;
    spare01 : BOOL ;
    StartOrder : BOOL ;
    CleareOrder : BOOL ;
    StopOrder : BOOL ;
    spare05 : BOOL ;
    spare06 : BOOL ;
    ReleaseOnline : BOOL ;
    Lifebit : BOOL ;
    spare11 : BOOL ;
    StartBasePos : BOOL ;
    ChangeOrder : BOOL ;
    QuitOrderFinished : BOOL ;
    ResetErrors : BOOL ;
    ServiceOn : BOOL ;
    BypassLimmitsOn : BOOL ;
    TotalLength : INT ;
    FaceLength : INT ;
    Circum : INT ;
    SourceBri : INT ;
    SourceTro : INT ;
    SourceLif : INT ;
    SourceTel : INT ;
    SourceAx04 : INT ;
    SourceAx05 : INT ;
    SourceAx06 : INT ;
    SourceAx07 : INT ;
    SourceAx08 : INT ;
    SourceAx09 : INT ;
    TargBri : INT ;
    TargTro : INT ;
    TargLif : INT ;
    TargTel : INT ;
    TargAx04 : INT ;
    TargAx05 : INT ;
    TargAx06 : INT ;
    TargAx07 : INT ;
    TargAx08 : INT ;
    TargAx09 : INT ;
    Occ00 : INT ;
    Occ01 : INT ;
    Occ02 : INT ;
    Occ03 : INT ;
    SafetyAreas00 : INT ;
    SafetyAreas01 : INT ;
    ParaCnt : INT ;
    ParaNo : INT ;
    ParaData : DINT ;
    _34 : INT ;
    _35 : INT ;
    _36 : INT ;
    _37 : INT ;
    _38 : INT ;
    _39 : INT ;
    _40 : INT ;
    _41 : INT ;
    _42 : INT ;
    _43 : INT ;
    _44 : INT ;
    CommCounterFromMaster : INT ;
    _46 : INT ;
    _47 : INT ;
    _48 : INT ;
    InvCrtWord : INT ;
    Bit100_0 : BOOL ;
    Bit100_1 : BOOL ;
    Bit100_2 : BOOL ;
    Bit100_3 : BOOL ;
    Bit100_4 : BOOL ;
    Bit100_5 : BOOL ;
    Bit00_6 : BOOL ;
    Bit100_7 : BOOL ;
    Release : BOOL ;
    BypassLimits : BOOL ;
    Service : BOOL ;
    Sw_Manual : BOOL ;
    Bit101_4 : BOOL ;
    Bit101_5 : BOOL ;
    Bit101_6 : BOOL ;
    Bit101_7 : BOOL ;
    BrPosRelease : INT ;
    TrPosRelease : INT ;
    LiPosRelease : INT ;
    TlPosRelease : INT ;
    spare_110 : INT ;
    spare_112 : INT ;
    spare_114 : INT ;
    spare_116 : INT ;
    spare_118 : INT ;
    spare_120 : INT ;
    spare_122 : INT ;
    spare_124 : INT ;
    spare_126 : INT ;
    Move : UDT 7;
    LS_1 : STRUCT
     Start_Load : BOOL ;
     Start_Unload : BOOL ;
     Step_Load : BOOL ;
     Step_Unload : BOOL ;
     CleareOrder : BOOL ;
     SPARE_05 : BOOL ;
     SPARE_06 : BOOL ;
     SPARE_07 : BOOL ;
     SPARE_10 : BOOL ;
     SPARE_11 : BOOL ;
     SPARE_12 : BOOL ;
     SPARE_13 : BOOL ;
     SPARE_14 : BOOL ;
     SPARE_15 : BOOL ;
     SPARE_16 : BOOL ;
     SPARE_17 : BOOL ;
     TotalLength : INT ;
     FaceLength : INT ;
     Circum : INT ;
    END_STRUCT ;
    Spare : ARRAY  [1 .. 19 ] OF WORD ;
   END_STRUCT ;
  END_STRUCT ;	
BEGIN
   TM.StateWord := 566;
   TM.BriActPos := 2;
   TM.TroActPos := 6;
   TM.LifActPos := 10;
   TM.TelActPos := 100;
   TM.BriMotorPos := L#4160;
   TM.TroMotorPos := L#16357;
   TM.LifMotorPos := L#4819;
   TM.TelMotorPos := L#10000;
   TM.CommCounterToMaster := 4664;
   TM.TeleskopsFree := TRUE;
   TM.Buffer_Free := TRUE;
   TM.Online := TRUE;
   TM.ReadyOnline := TRUE;
   TM.TeleskopCenterpos := TRUE;
   TM.Move.Action := 3;
   TM.Move.Value_01 := 2;
   TM.Move.Value_02 := 6;
   TM.Move.Value_03 := 10;
   TM.Move.Value_04 := 100;
   TM.LS_1.Online := TRUE;
   TM.LS_1.Ready := TRUE;
   TM.LS_1.Palette_In_Station := TRUE;
   TM.LS_1.Pos_11_Free := TRUE;
   TM.LS_1.Pos_12_Free := TRUE;
   TM.LS_2.Online := TRUE;
   TM.LS_2.Ready := TRUE;
   TM.LS_2.Palette_In_Station := TRUE;
   TM.LS_2.Pos_11_Free := TRUE;
   TM.LS_2.Pos_12_Free := TRUE;
   TM.LS_3.Online := TRUE;
   TM.LS_3.Ready := TRUE;
   TM.LS_3.Palette_In_Station := TRUE;
   TM.LS_3.Pos_11_Free := TRUE;
   TM.LS_3.Pos_12_Free := TRUE;
   TM.Spare[1] := W#16#4241;
   TM.Spare[2] := W#16#5545;
   TM.Spare[3] := W#16#5520;
   FM.TotalLength := 2090;
   FM.FaceLength := 1499;
   FM.Circum := 784;
   FM.SourceBri := 99;
   FM.SourceTro := 99;
   FM.SourceLif := 1;
   FM.SourceTel := 1;
   FM.TargBri := 2;
   FM.TargTro := 6;
   FM.TargLif := 10;
   FM.TargTel := 1;
   FM.ParaCnt := 321;
   FM.ParaNo := 654;
   FM.ParaData := L#76542;
   FM.CommCounterFromMaster := 4663;
   FM.Bit100_1 := TRUE;
   FM.Bit100_2 := TRUE;
   FM.Move.MsgCounter := 751;
   FM.Move.Action := 3;
   FM.Move.Value_01 := 2;
   FM.Move.Value_02 := 6;
   FM.Move.Value_03 := 10;
   FM.Move.Value_04 := 100;
END_DATA_BLOCK

DATA_BLOCK "BRI_Positions"	// DB 200
VERSION : 0.1
  STRUCT
   BRIPos : ARRAY  [0 .. 101 ] OF STRUCT
    No : INT ;	//number of position
    Val_BRI : DINT ;	//value of bridge position
    Val_TRO : DINT ;	//value of trolley position
    DB_No : INT ;	//Hook DB-Number
    DB_No_2 : INT ;	//Hook DB-Number 2
   END_STRUCT ;
   di_BRI_Pos : DINT ;
   di_TRO_Pos : DINT ;
  END_STRUCT ;	
BEGIN
   BRIPos[0].No := 1;
   BRIPos[0].Val_BRI := L#37007;
   BRIPos[1].No := 2;
   BRIPos[1].Val_BRI := L#33953;
   BRIPos[2].No := 3;
   BRIPos[2].Val_BRI := L#30903;
   BRIPos[3].No := 4;
   BRIPos[3].Val_BRI := L#27852;
   BRIPos[4].No := 5;
   BRIPos[4].Val_BRI := L#24802;
   BRIPos[5].No := 6;
   BRIPos[5].Val_BRI := L#19152;
   BRIPos[6].No := 7;
   BRIPos[6].Val_BRI := L#16097;
   BRIPos[7].No := 8;
   BRIPos[7].Val_BRI := L#13044;
   BRIPos[8].No := 9;
   BRIPos[8].Val_BRI := L#9996;
   BRIPos[9].No := 10;
   BRIPos[9].Val_BRI := L#6945;
   BRIPos[10].No := 11;
   BRIPos[10].Val_BRI := L#3442;
END_DATA_BLOCK

DATA_BLOCK "ProfiNET"	// DB 400
VERSION : 0.0
  STRUCT
   STAT0 : ARRAY  [-32768 .. -31295 ] OF BYTE ;
  END_STRUCT ;	
BEGIN
   STAT0[-32745] := B#16#1;
   STAT0[-32743] := B#16#1;
   STAT0[-32741] := B#16#1;
   STAT0[-31744] := B#16#90;
   STAT0[-31743] := B#16#1;
   STAT0[-31742] := B#16#1;
   STAT0[-31737] := B#16#2;
END_DATA_BLOCK

DATA_BLOCK "Error_Safety"	// DB 410
AUTHOR : Koenig
VERSION : 0.1
  STRUCT
   Error_09 : BOOL ;
   Error_10 : BOOL ;
   Error_11 : BOOL ;
   Error_12 : BOOL ;
   Error_13 : BOOL ;
   Error_14 : BOOL ;
   Error_15 : BOOL ;
   Error_16 : BOOL ;
   Error_01 : BOOL ;	//Wago unit #1 disturbed
   Error_02 : BOOL ;	//Wago unit #2 disturbed
   Error_03 : BOOL ;	//Wago unit #3 disturbed
   Error_04 : BOOL ;
   Error_05 : BOOL ;
   Error_06 : BOOL ;	//ESTOP active
   Error_07 : BOOL ;	//Actual position invalid
   Error_08 : BOOL ;	//Actual position not in work area
   Error_25 : BOOL ;
   Error_26 : BOOL ;
   Error_27 : BOOL ;
   Error_28 : BOOL ;
   Error_29 : BOOL ;
   Error_30 : BOOL ;
   Error_31 : BOOL ;
   Error_32 : BOOL ;
   Error_17 : BOOL ;
   Error_18 : BOOL ;
   Error_19 : BOOL ;
   Error_20 : BOOL ;
   Error_21 : BOOL ;
   Error_22 : BOOL ;
   Error_23 : BOOL ;
   Error_24 : BOOL ;
   Error_41 : BOOL ;
   Error_42 : BOOL ;
   Error_43 : BOOL ;
   Error_44 : BOOL ;
   Error_45 : BOOL ;
   Error_46 : BOOL ;
   Error_47 : BOOL ;
   Error_48 : BOOL ;
  END_STRUCT ;	
BEGIN
END_DATA_BLOCK

// DB 415: know-how protected block, not included

// DB 545: know-how protected block, not included

// DB 546: know-how protected block, not included

// DB 547: know-how protected block, not included

// DB 548: know-how protected block, not included

// DB 549: know-how protected block, not included

// DB 550: know-how protected block, not included

// DB 551: know-how protected block, not included

// DB 552: know-how protected block, not included

// DB 553: know-how protected block, not included

// DB 554: know-how protected block, not included

// DB 555: know-how protected block, not included

// DB 556: know-how protected block, not included

// DB 557: know-how protected block, not included

// DB 558: know-how protected block, not included

DATA_BLOCK "F_IO"	// DB 690
AUTHOR : Koenig
VERSION : 0.1
  STRUCT
   BRI_EStop : BOOL ;
   BRI_FB_FastStop : BOOL ;
   BRI_FB_EStop_CH1 : BOOL ;
   BRI_FB_EStop_CH2 : BOOL ;
   BRI_Input_04 : BOOL ;
   BRI_Input_05 : BOOL ;
   BRI_Input_06 : BOOL ;
   BRI_Input_07 : BOOL ;
   BRI_TRO_inParkPos_CH1 : BOOL ;
   BRI_TRO_inParkPos_CH2 : BOOL ;
   BRI_Brake_OK : BOOL ;
   BRI_Input_11 : BOOL ;
   BRI_Input_12 : BOOL ;
   BRI_Input_13 : BOOL ;
   BRI_Input_14 : BOOL ;
   BRI_HardwareOK : BOOL ;
   TRO_FB_Bypass_RC : BOOL ;
   TRO_Spare_DI_35_1 : BOOL ;
   TRO_FB_Estop_Lift : BOOL ;
   TRO_FB_Estop_TRO : BOOL ;
   TRO_FB_Telescope : BOOL ;
   TRO_Spare_DI_40_1 : BOOL ;
   TRO_FB_Estop_CH1 : BOOL ;
   TRO_FB_Estop_CH2 : BOOL ;
   TRO_EStop : BOOL ;
   TRO_Spare_DI_45_1 : BOOL ;
   TRO_Spare_DI_45_2 : BOOL ;
   TRO_BrakesOK : BOOL ;
   TRO_Input_12 : BOOL ;
   TRO_Input_13 : BOOL ;
   TRO_Input_14 : BOOL ;
   TRO_HardwareOK : BOOL ;
   LIF_Input_00 : BOOL ;
   LIF_Input_01 : BOOL ;
   LIF_Input_02 : BOOL ;
   LIF_Input_03 : BOOL ;
   LIF_Input_04 : BOOL ;
   LIF_Input_05 : BOOL ;
   LIF_Input_06 : BOOL ;
   LIF_Input_07 : BOOL ;
   LIF_Input_08 : BOOL ;
   LIF_Input_09 : BOOL ;
   LIF_Input_10 : BOOL ;
   LIF_Input_11 : BOOL ;
   LIF_Input_12 : BOOL ;
   LIF_Input_13 : BOOL ;
   LIF_Input_14 : BOOL ;
   LIF_HardwareOK : BOOL ;
   CB1_FastStop_Gate_CH1 : BOOL ;
   CB1_FastStop_Gate_CH2 : BOOL ;
   CB1_SPARE_DI220_2 : BOOL ;
   CB1_SPARE_DI220_3 : BOOL ;
   CB1_SPARE_DI225_0 : BOOL ;
   CB1_FastStop : BOOL ;
   CB1_Mode_Auto : BOOL ;
   CB1_Mode_Service : BOOL ;
   CB1_LS1_Door_CH1 : BOOL ;
   CB1_LS1_Door_CH2 : BOOL ;
   CB1_LS2_Door_CH1 : BOOL ;
   CB1_LS2_Door_CH2 : BOOL ;
   CB1_LS3_Door_CH1 : BOOL ;
   CB1_LS3_Door_CH2 : BOOL ;
   CB1_ServiceDoor1_CH1 : BOOL ;
   CB1_ServiceDoor1_CH2 : BOOL ;
   CB1_ServiceDoor2_CH1 : BOOL ;
   CB1_ServiceDoor2_CH2 : BOOL ;
   CB1_ServiceDoor3_CH1 : BOOL ;
   CB1_ServiceDoor3_CH2 : BOOL ;
   CB1_ServiceDoor4_CH1 : BOOL ;
   CB1_ServiceDoor4_CH2 : BOOL ;
   CB1_EStop_Buttons_CH1 : BOOL ;
   CB1_EStop_Buttons_CH2 : BOOL ;
   CB1_EStop_Doors_CH1 : BOOL ;
   CB1_EStop_Doors_CH2 : BOOL ;
   CB1_Service_CH1 : BOOL ;
   CB1_Service_CH2 : BOOL ;
   CB1_Bypass_CH1 : BOOL ;
   CB1_Bypass_CH2 : BOOL ;
   CB1_Auto_ON : BOOL ;
   CB1_SPARE_DI240_7 : BOOL ;
   CB1_PowerON_1 : BOOL ;
   CB1_PowerON_2 : BOOL ;
   CB1_SPARE_DO220_2 : BOOL ;
   CB1_SPARE_DO220_3 : BOOL ;
   CB1_SPARE_DO225_0 : BOOL ;
   CB1_SPARE_DO225_1 : BOOL ;
   CB1_SPARE_DO225_2 : BOOL ;
   CB1_SPARE_DO225_3 : BOOL ;
   MB1_Power_ON_1 : BOOL ;
   MB1_Power_ON_2 : BOOL ;
   MB1_ESTOP_1 : BOOL ;
   MB1_ESTOP_2 : BOOL ;
   MB1_HardwareOK : BOOL ;
   MB1_FB_Power_ON : BOOL ;
   MB1_INPUT_07 : BOOL ;
   MB1_INPUT_08 : BOOL ;
   SU1_HardwareOK : BOOL ;
   SU1_Scanner_Plus_OK : BOOL ;
   SU1_Scanner_Minus_OK : BOOL ;
   SU1_ReglerPowerON : BOOL ;
   SU1_INPUT_05 : BOOL ;
   SU1_INPUT_06 : BOOL ;
   SU1_INPUT_07 : BOOL ;
   SU1_INPUT_08 : BOOL ;
   SU2_HardwareOK : BOOL ;
   SU2_Scanner_Plus_OK : BOOL ;
   SU2_Scanner_Minus_OK : BOOL ;
   SU2_ReglerPowerON : BOOL ;
   SU2_INPUT_05 : BOOL ;
   SU2_INPUT_06 : BOOL ;
   SU2_INPUT_07 : BOOL ;
   SU2_INPUT_08 : BOOL ;
  END_STRUCT ;	
BEGIN
   BRI_Input_04 := TRUE;
   TRO_FB_Bypass_RC := TRUE;
   TRO_FB_Estop_TRO := TRUE;
   TRO_FB_Telescope := TRUE;
   LIF_Input_00 := TRUE;
   CB1_Mode_Auto := TRUE;
   CB1_EStop_Buttons_CH2 := TRUE;
   CB1_EStop_Doors_CH1 := TRUE;
   CB1_EStop_Doors_CH2 := TRUE;
   CB1_Service_CH1 := TRUE;
   CB1_Service_CH2 := TRUE;
   CB1_Auto_ON := TRUE;
   CB1_SPARE_DI240_7 := TRUE;
   CB1_PowerON_1 := TRUE;
   CB1_PowerON_2 := TRUE;
   CB1_SPARE_DO220_2 := TRUE;
   CB1_SPARE_DO220_3 := TRUE;
   CB1_SPARE_DO225_0 := TRUE;
   CB1_SPARE_DO225_1 := TRUE;
   CB1_SPARE_DO225_2 := TRUE;
   CB1_SPARE_DO225_3 := TRUE;
   MB1_FB_Power_ON := TRUE;
END_DATA_BLOCK

DATA_BLOCK "F_GBL_RECV"	// DB 750
AUTHOR : Koenig
FAMILY : COM_DBS7
VERSION : 0.1
  STRUCT
   Signal01 : BOOL ;	//Automatic mode
   Signal02 : BOOL ;	//Bypass
   Signal03 : BOOL ;	//Reset
   Signal04 : BOOL ;	//NO E-Stop
   Signal05 : BOOL ;	//Start Automatic
   Signal06 : BOOL ;	//Release drive
   Signal07 : BOOL ;	//Release fast drive
   Signal08 : BOOL ;	//Service mode
   Signal09 : BOOL ;
   Signal10 : BOOL ;
   Signal11 : BOOL ;
   Signal12 : BOOL ;
   Signal13 : BOOL ;
   Signal14 : BOOL ;
   Signal15 : BOOL ;
   Signal16 : BOOL ;
   Signal17 : BOOL ;
   Signal18 : BOOL ;
   Signal19 : BOOL ;
   Signal20 : BOOL ;
   Signal21 : BOOL ;
   Signal22 : BOOL ;
   Signal23 : BOOL ;
   Signal24 : BOOL ;
   Signal25 : BOOL ;
   Signal26 : BOOL ;
   Signal27 : BOOL ;
   Signal28 : BOOL ;
   Signal29 : BOOL ;
   Signal30 : BOOL ;
   Signal31 : BOOL ;
   Signal32 : BOOL ;
   Value01 : INT ;
   Value02 : INT ;
   Value03 : INT ;
   Value04 : INT ;
  END_STRUCT ;	
BEGIN
   Signal01 := TRUE;
   Signal04 := TRUE;
   Signal06 := TRUE;
   Signal10 := TRUE;
   Signal32 := TRUE;
END_DATA_BLOCK

// DB 751: know-how protected block, not included

DATA_BLOCK "F_GBL_SEND"	// DB 752
AUTHOR : Koenig
FAMILY : COM_DBS7
VERSION : 0.1
  STRUCT
   Signal01 : BOOL ;
   Signal02 : BOOL ;
   Signal03 : BOOL ;
   Signal04 : BOOL ;
   Signal05 : BOOL ;
   Signal06 : BOOL ;
   Signal07 : BOOL ;
   Signal08 : BOOL ;
   Signal09 : BOOL ;
   Signal10 : BOOL ;
   Signal11 : BOOL ;
   Signal12 : BOOL ;
   Signal13 : BOOL ;
   Signal14 : BOOL ;
   Signal15 : BOOL ;
   Signal16 : BOOL ;
   Value01 : INT ;
   Value02 : INT ;
   Value03 : INT ;
  END_STRUCT ;	
BEGIN
   Value01 := 3395;
   Value03 := 2;
END_DATA_BLOCK

// DB 753: know-how protected block, not included

DATA_BLOCK "IDB_WagoiPar_BRI"	// DB 920
AUTHOR : JPR
FAMILY : WAGOiPar
VERSION : 0.0
"WAGO_iPar_UDL_4_Mod"
BEGIN
END_DATA_BLOCK

DATA_BLOCK "DB_iPar_Diag"	// DB 930
AUTHOR : JPR
FAMILY : WAGOiPar
VERSION : 0.0
"DiagPROFIsafe_V2_iPar"
BEGIN
END_DATA_BLOCK

DATA_BLOCK "iPar_Data_Bridge"	// DB 1920
TITLE = Vorlage Datenbaustein zur Ablage der iParameter für FB37
//Template data block used in combination with FB37
//
AUTHOR : JPR
FAMILY : WAGOiPar
NAME : iParUDL4
VERSION : 5.1
  STRUCT
   versionInfo_1 : INT  := 37;	//version info main
   versionInfo_2 : WORD  := W#16#501;	//version info release
   chkInfoData : WORD ;	//check info data
   fctReqTimeout : INT  := 6000;	//function request timeout (default 6000; av.cycle plc 5 ms - timeout 30 s)
   maxModules : INT  := 1;	//amount PROFIsafe modules FB41
   type_module_1 : INT ;	//type module 1 (661/662/663/666/667/669)
   adr_module_1 : INT ;	//I/O address module 1
   bussystem_mod_1 : INT ;	//used bussystem module 1 (0 = DP / 1 = PN)
   type_module_2 : INT ;	//type module 2 (661/662/663/666/667/669)
   adr_module_2 : INT ;	//I/O address module 2
   bussystem_mod_2 : INT ;	//used bussystem module 2 (0 = DP / 1 = PN)
   type_module_3 : INT ;	//type module 3 (661/662/663/666/667/669)
   adr_module_3 : INT ;	//I/O address module 3
   bussystem_mod_3 : INT ;	//used bussystem module 3 (0 = DP / 1 = PN)
   type_module_4 : INT ;	//type module 4 (661/662/663/666/667/669)
   adr_module_4 : INT ;	//I/O address module 4
   bussystem_mod_4 : INT ;	//used bussystem module 4 (0 = DP / 1 = PN)
   spare_34 : WORD ;
   spare_36 : WORD ;
   spare_38 : WORD ;
   spare_40 : WORD ;
   spare_42 : WORD ;
   spare_44 : WORD ;
   spare_46 : WORD ;
   spare_48 : WORD ;
   spare_50 : WORD ;
   spare_52 : WORD ;
   spare_54 : WORD ;
   spare_56 : WORD ;
   spare_58 : WORD ;
   spare_60 : WORD ;
   spare_62 : WORD ;
   spare_64 : WORD ;
   spare_66 : WORD ;
   spare_68 : WORD ;
   spare_70 : WORD ;
   spare_72 : WORD ;
   spare_74 : WORD ;
   spare_76 : WORD ;
   spare_78 : WORD ;
   spare_80 : WORD ;
   resFctReq_ok : DWORD ;	//response function request ok - "bit per module"
   resFctReq_error : DWORD ;	//response function request error - "bit per module"
   startupDate : DATE ;	//startup date application slave
   startupTime : TIME_OF_DAY ;	//startup time application slave
   slaveConfigInfo : DWORD ;	//info available PROFIsafe modules at slave
   QBAD_moduleActive : DWORD ;	//info QBAD at PROFIsafe module active
   ACK_REQ_moduleActive : DWORD ;	//info ACK_REQ at PROFIsafe module active
   READ_DIAG_REQ_module : DWORD ;	//info READ_DIAG_REQ at PROFIsafe module active
   init_fb_done : DWORD ;	//info init FB done
   check_cfg_done : DWORD ;	//info check cfg done
   upload_done : DWORD ;	//info upload slave done
   download_done : DWORD ;	//info download slave done
   compare_done : DWORD ;	//info compare slave done
   actDateCyle : DATE ;	//actual system date of cycle
   actTimeCyle : TIME_OF_DAY ;	//actual system time of cycle
   cmdCtrl_FB37 : WORD ;	//cmd / ctrl information FB37
   comCountStart_1 : WORD ;	//comCountStart indication 1
   mod_type_1 : WORD ;	//module type 1
   mod_version_1 : WORD ;	//module version 1
   spare_146 : WORD ;
   spare_148 : WORD ;
   upl_date_mod_1 : DATE ;	//upload date module 1
   upl_time_mod_1 : TIME_OF_DAY ;	//upload time module 1
   dnl_date_mod_1 : DATE ;	//download date module 1
   dnl_time_mod_1 : TIME_OF_DAY ;	//download time module 1
   cmp_date_mod_1 : DATE ;	//compare date module 1
   cmp_time_mod_1 : TIME_OF_DAY ;	//compare time module 1
   dsv_info_mod_1 : WORD ;	//dataset info module 1
   data_0_mod_1 : WORD ;	//data 0 - 1 module 1
   data_2_mod_1 : WORD ;	//data 2 - 3 module 1
   data_4_mod_1 : WORD ;	//data 4 - 5 module 1
   data_6_mod_1 : WORD ;	//data 6 - 7 module 1
   data_8_mod_1 : WORD ;	//data 8 - 9 module 1
   data_10_mod_1 : WORD ;	//data 10 - 11 module 1
   data_12_mod_1 : WORD ;	//data 12 - 13 module 1
   data_14_mod_1 : WORD ;	//data 14 - 15 module 1
   data_16_mod_1 : WORD ;	//data 16 - 17 module 1
   data_18_mod_1 : WORD ;	//data 18 - 19 module 1
   data_20_mod_1 : WORD ;	//data 20 - 21 module 1
   data_22_mod_1 : WORD ;	//data 22 - 23 module 1
   data_24_mod_1 : WORD ;	//data 24 - 25 module 1
   data_26_mod_1 : WORD ;	//data 26 - 27 module 1
   data_28_mod_1 : WORD ;	//data 28 - 29 module 1
   data_30_mod_1 : WORD ;	//data 30 - 31 module 1
   data_32_mod_1 : WORD ;	//data 32 - 33 module 1
   data_34_mod_1 : WORD ;	//data 34 - 35 module 1
   data_36_mod_1 : WORD ;	//data 36 - 37 module 1
   data_38_mod_1 : WORD ;	//data 38 - 39 module 1
   spare_210 : WORD ;
   spare_212 : WORD ;
   spare_214 : WORD ;
   spare_216 : WORD ;
   spare_218 : WORD ;
   error_Com_1 : WORD ;	//error indication  Com  module 1
   error_nb_Com_1 : WORD ;	//error number indication  Com  module 1
   state_SFB52a_1 : WORD ;	//state SFB52 part 1 module 1
   state_SFB52b_1 : WORD ;	//state SFB52 part 2 module 1
   state_SFB53a_1 : WORD ;	//state SFB53 part 1 module 1
   state_SFB53b_1 : WORD ;	//state SFB53 part 2 module 1
   spare_232 : WORD ;
   error_date_mod_1 : DATE ;	//error date module 1
   error_time_mod_1 : TIME_OF_DAY ;	//error time module 1
   error_info_mod_1 : WORD ;	//error info read values module 1
   error_F_Module_mod_1 : WORD ;	//error safety module module 1
   error_F_DI_1_mod_1 : WORD ;	//error safety input 1 module 1
   error_F_DI_2_mod_1 : WORD ;	//error safety input 2 module 1
   error_F_DI_3_mod_1 : WORD ;	//error safety input 3 module 1
   error_F_DI_4_mod_1 : WORD ;	//error safety input 4 module 1
   error_F_DI_5_mod_1 : WORD ;	//error safety input 5 module 1
   error_F_DI_6_mod_1 : WORD ;	//error safety input 6 module 1
   error_F_DI_7_mod_1 : WORD ;	//error safety input 7 module 1
   error_F_DI_8_mod_1 : WORD ;	//error safety input 8 module 1
   error_F_DO_1_mod_1 : WORD ;	//error safety output 1 module 1
   error_F_DO_2_mod_1 : WORD ;	//error safety output 2 module 1
   error_F_DO_3_mod_1 : WORD ;	//error safety output 3 module 1
   error_F_DO_4_mod_1 : WORD ;	//error safety output 4 module 1
   error_Reg52_mod_1 : WORD ;	//error safety module register 52 module 1
   error_Reg53_mod_1 : WORD ;	//error safety module register 53 module 1
   error_Reg54_mod_1 : WORD ;	//error safety module register 54 module 1
   error_Reg55_mod_1 : WORD ;	//error safety module register 55 module 1
   spare_276 : WORD ;
   spare_278 : WORD ;
   comCountStart_2 : WORD ;	//comCountStart indication 2
   mod_type_2 : WORD ;	//module type 2
   mod_version_2 : WORD ;	//module version 2
   spare_286 : WORD ;
   spare_288 : WORD ;
   upl_date_mod_2 : DATE ;	//upload date module 2
   upl_time_mod_2 : TIME_OF_DAY ;	//upload time module 2
   dnl_date_mod_2 : DATE ;	//download date module 2
   dnl_time_mod_2 : TIME_OF_DAY ;	//download time module 2
   cmp_date_mod_2 : DATE ;	//compare date module 2
   cmp_time_mod_2 : TIME_OF_DAY ;	//compare time module 2
   dsv_info_mod_2 : WORD ;	//dataset info module 2
   data_0_mod_2 : WORD ;	//data 0 - 1 module 2
   data_2_mod_2 : WORD ;	//data 2 - 3 module 2
   data_4_mod_2 : WORD ;	//data 4 - 5 module 2
   data_6_mod_2 : WORD ;	//data 6 - 7 module 2
   data_8_mod_2 : WORD ;	//data 8 - 9 module 2
   data_10_mod_2 : WORD ;	//data 10 - 11 module 2
   data_12_mod_2 : WORD ;	//data 12 - 13 module 2
   data_14_mod_2 : WORD ;	//data 14 - 15 module 2
   data_16_mod_2 : WORD ;	//data 16 - 17 module 2
   data_18_mod_2 : WORD ;	//data 18 - 19 module 2
   data_20_mod_2 : WORD ;	//data 20 - 21 module 2
   data_22_mod_2 : WORD ;	//data 22 - 23 module 2
   data_24_mod_2 : WORD ;	//data 24 - 25 module 2
   data_26_mod_2 : WORD ;	//data 26 - 27 module 2
   data_28_mod_2 : WORD ;	//data 28 - 29 module 2
   data_30_mod_2 : WORD ;	//data 30 - 31 module 2
   data_32_mod_2 : WORD ;	//data 32 - 33 module 2
   data_34_mod_2 : WORD ;	//data 34 - 35 module 2
   data_36_mod_2 : WORD ;	//data 36 - 37 module 2
   data_38_mod_2 : WORD ;	//data 38 - 39 module 2
   spare_350 : WORD ;
   spare_352 : WORD ;
   spare_354 : WORD ;
   spare_356 : WORD ;
   spare_358 : WORD ;
   error_Com_2 : WORD ;	//error indication  Com  module 2
   error_nb_Com_2 : WORD ;	//error number indication  Com  module 2
   state_SFB52a_2 : WORD ;	//state SFB52 part 1 module 2
   state_SFB52b_2 : WORD ;	//state SFB52 part 2 module 2
   state_SFB53a_2 : WORD ;	//state SFB53 part 1 module 2
   state_SFB53b_2 : WORD ;	//state SFB53 part 2 module 2
   spare_372 : WORD ;
   error_date_mod_2 : DATE ;	//error date module 2
   error_time_mod_2 : TIME_OF_DAY ;	//error time module 2
   error_info_mod_2 : WORD ;	//error info read values module 2
   error_F_Module_mod_2 : WORD ;	//error safety module module 2
   error_F_DI_1_mod_2 : WORD ;	//error safety input 1 module 2
   error_F_DI_2_mod_2 : WORD ;	//error safety input 2 module 2
   error_F_DI_3_mod_2 : WORD ;	//error safety input 3 module 2
   error_F_DI_4_mod_2 : WORD ;	//error safety input 4 module 2
   error_F_DI_5_mod_2 : WORD ;	//error safety input 5 module 2
   error_F_DI_6_mod_2 : WORD ;	//error safety input 6 module 2
   error_F_DI_7_mod_2 : WORD ;	//error safety input 7 module 2
   error_F_DI_8_mod_2 : WORD ;	//error safety input 8 module 2
   error_F_DO_1_mod_2 : WORD ;	//error safety output 1 module 2
   error_F_DO_2_mod_2 : WORD ;	//error safety output 2 module 2
   error_F_DO_3_mod_2 : WORD ;	//error safety output 3 module 2
   error_F_DO_4_mod_2 : WORD ;	//error safety output 4 module 2
   error_Reg52_mod_2 : WORD ;	//error safety module register 52 module 2
   error_Reg53_mod_2 : WORD ;	//error safety module register 53 module 2
   error_Reg54_mod_2 : WORD ;	//error safety module register 54 module 2
   error_Reg55_mod_2 : WORD ;	//error safety module register 55 module 2
   spare_416 : WORD ;
   spare_418 : WORD ;
   comCountStart_3 : WORD ;	//comCountStart indication 3
   mod_type_3 : WORD ;	//module type 3
   mod_version_3 : WORD ;	//module version 3
   spare_426 : WORD ;
   spare_428 : WORD ;
   upl_date_mod_3 : DATE ;	//upload date module 3
   upl_time_mod_3 : TIME_OF_DAY ;	//upload time module 3
   dnl_date_mod_3 : DATE ;	//download date module 3
   dnl_time_mod_3 : TIME_OF_DAY ;	//download time module 3
   cmp_date_mod_3 : DATE ;	//compare date module  3
   cmp_time_mod_3 : TIME_OF_DAY ;	//compare time module  3
   dsv_info_mod_3 : WORD ;	//dataset info module 3
   data_0_mod_3 : WORD ;	//data 0 - 1 module 3
   data_2_mod_3 : WORD ;	//data 2 - 3 module 3
   data_4_mod_3 : WORD ;	//data 4 - 5 module 3
   data_6_mod_3 : WORD ;	//data 6 - 7 module 3
   data_8_mod_3 : WORD ;	//data 8 - 9 module 3
   data_10_mod_3 : WORD ;	//data 10 - 11 module 3
   data_12_mod_3 : WORD ;	//data 12 - 13 module 3
   data_14_mod_3 : WORD ;	//data 14 - 15 module 3
   data_16_mod_3 : WORD ;	//data 16 - 17 module 3
   data_18_mod_3 : WORD ;	//data 18 - 19 module 3
   data_20_mod_3 : WORD ;	//data 20 - 21 module 3
   data_22_mod_3 : WORD ;	//data 22 - 23 module 3
   data_24_mod_3 : WORD ;	//data 24 - 25 module 3
   data_26_mod_3 : WORD ;	//data 26 - 27 module 3
   data_28_mod_3 : WORD ;	//data 28 - 29 module 3
   data_30_mod_3 : WORD ;	//data 30 - 31 module 3
   data_32_mod_3 : WORD ;	//data 32 - 33 module 3
   data_34_mod_3 : WORD ;	//data 34 - 35 module 3
   data_36_mod_3 : WORD ;	//data 36 - 37 module 3
   data_38_mod_3 : WORD ;	//data 38 - 39 module 3
   spare_490 : WORD ;
   spare_492 : WORD ;
   spare_494 : WORD ;
   spare_496 : WORD ;
   spare_498 : WORD ;
   error_Com_3 : WORD ;	//error indication  Com  module 3
   error_nb_Com_3 : WORD ;	//error number indication  Com  module 3
   state_SFB52a_3 : WORD ;	//state SFB52 part 1 module 3
   state_SFB52b_3 : WORD ;	//state SFB52 part 2 module 3
   state_SFB53a_3 : WORD ;	//state SFB53 part 1 module 3
   state_SFB53b_3 : WORD ;	//state SFB53 part 2 module 3
   spare_512 : WORD ;
   error_date_mod_3 : DATE ;	//error date module 3
   error_time_mod_3 : TIME_OF_DAY ;	//error time module 3
   error_info_mod_3 : WORD ;	//error info read values module 3
   error_F_Module_mod_3 : WORD ;	//error safety module module 3
   error_F_DI_1_mod_3 : WORD ;	//error safety input 1 module 3
   error_F_DI_2_mod_3 : WORD ;	//error safety input 2 module 3
   error_F_DI_3_mod_3 : WORD ;	//error safety input 3 module 3
   error_F_DI_4_mod_3 : WORD ;	//error safety input 4 module 3
   error_F_DI_5_mod_3 : WORD ;	//error safety input 5 module 3
   error_F_DI_6_mod_3 : WORD ;	//error safety input 6 module 3
   error_F_DI_7_mod_3 : WORD ;	//error safety input 7 module 3
   error_F_DI_8_mod_3 : WORD ;	//error safety input 8 module 3
   error_F_DO_1_mod_3 : WORD ;	//error safety output 1 module 3
   error_F_DO_2_mod_3 : WORD ;	//error safety output 2 module 3
   error_F_DO_3_mod_3 : WORD ;	//error safety output 3 module 3
   error_F_DO_4_mod_3 : WORD ;	//error safety output 4 module 3
   error_Reg52_mod_3 : WORD ;	//error safety module register 52 module 3
   error_Reg53_mod_3 : WORD ;	//error safety module register 53 module 3
   error_Reg54_mod_3 : WORD ;	//error safety module register 54 module 3
   error_Reg55_mod_3 : WORD ;	//error safety module register 55 module 3
   spare_556 : WORD ;
   spare_558 : WORD ;
   comCountStart_4 : WORD ;	//comCountStart indication 4
   mod_type_4 : WORD ;	//module type  4
   mod_version_4 : WORD ;	//module version  4
   spare_566 : WORD ;
   spare_568 : WORD ;
   upl_date_mod_4 : DATE ;	//upload date module  4
   upl_time_mod_4 : TIME_OF_DAY ;	//upload time module  4
   dnl_date_mod_4 : DATE ;	//download date module  4
   dnl_time_mod_4 : TIME_OF_DAY ;	//download time module  4
   cmp_date_mod_4 : DATE ;	//compare date module   4
   cmp_time_mod_4 : TIME_OF_DAY ;	//compare time module   4
   dsv_info_mod_4 : WORD ;	//dataset info module 4
   data_0_mod_4 : WORD ;	//data 0 - 1 module  4
   data_2_mod_4 : WORD ;	//data 2 - 3 module  4
   data_4_mod_4 : WORD ;	//data 4 - 5 module  4
   data_6_mod_4 : WORD ;	//data 6 - 7 module  4
   data_8_mod_4 : WORD ;	//data 8 - 9 module  4
   data_10_mod_4 : WORD ;	//data 10 - 11 module  4
   data_12_mod_4 : WORD ;	//data 12 - 13 module  4
   data_14_mod_4 : WORD ;	//data 14 - 15 module  4
   data_16_mod_4 : WORD ;	//data 16 - 17 module  4
   data_18_mod_4 : WORD ;	//data 18 - 19 module  4
   data_20_mod_4 : WORD ;	//data 20 - 21 module  4
   data_22_mod_4 : WORD ;	//data 22 - 23 module  4
   data_24_mod_4 : WORD ;	//data 24 - 25 module  4
   data_26_mod_4 : WORD ;	//data 26 - 27 module  4
   data_28_mod_4 : WORD ;	//data 28 - 29 module  4
   data_30_mod_4 : WORD ;	//data 30 - 31 module  4
   data_32_mod_4 : WORD ;	//data 32 - 33 module  4
   data_34_mod_4 : WORD ;	//data 34 - 35 module  4
   data_36_mod_4 : WORD ;	//data 36 - 37 module  4
   data_38_mod_4 : WORD ;	//data 38 - 39 module  4
   spare_630 : WORD ;
   spare_632 : WORD ;
   spare_634 : WORD ;
   spare_636 : WORD ;
   spare_638 : WORD ;
   error_Com_4 : WORD ;	//error indication  Com  module 4
   error_nb_Com_4 : WORD ;	//error number indication  Com  module 4
   state_SFB52a_4 : WORD ;	//state SFB52 part 1 module 4
   state_SFB52b_4 : WORD ;	//state SFB52 part 2 module 4
   state_SFB53a_4 : WORD ;	//state SFB53 part 1 module 4
   state_SFB53b_4 : WORD ;	//state SFB53 part 2 module 4
   spare_652 : WORD ;
   error_date_mod_4 : DATE ;	//error date module 4
   error_time_mod_4 : TIME_OF_DAY ;	//error time module 4
   error_info_mod_4 : WORD ;	//error info read values module 4
   error_F_Module_mod_4 : WORD ;	//error safety module module 4
   error_F_DI_1_mod_4 : WORD ;	//error safety input 1 module 4
   error_F_DI_2_mod_4 : WORD ;	//error safety input 2 module 4
   error_F_DI_3_mod_4 : WORD ;	//error safety input 3 module 4
   error_F_DI_4_mod_4 : WORD ;	//error safety input 4 module 4
   error_F_DI_5_mod_4 : WORD ;	//error safety input 5 module 4
   error_F_DI_6_mod_4 : WORD ;	//error safety input 6 module 4
   error_F_DI_7_mod_4 : WORD ;	//error safety input 7 module 4
   error_F_DI_8_mod_4 : WORD ;	//error safety input 8 module 4
   error_F_DO_1_mod_4 : WORD ;	//error safety output 1 module 4
   error_F_DO_2_mod_4 : WORD ;	//error safety output 2 module 4
   error_F_DO_3_mod_4 : WORD ;	//error safety output 3 module 4
   error_F_DO_4_mod_4 : WORD ;	//error safety output 4 module 4
   error_Reg52_mod_4 : WORD ;	//error safety module register 52 module 4
   error_Reg53_mod_4 : WORD ;	//error safety module register 53 module 4
   error_Reg54_mod_4 : WORD ;	//error safety module register 54 module 4
   error_Reg55_mod_4 : WORD ;	//error safety module register 55 module 4
   spare_696 : WORD ;
   spare_698 : WORD ;
  END_STRUCT ;	
BEGIN
   versionInfo_1 := 37;
   versionInfo_2 := W#16#501;
   chkInfoData := W#16#2;
   fctReqTimeout := 6000;
   maxModules := 2;
   type_module_1 := 667;
   adr_module_1 := 20;
   bussystem_mod_1 := 1;
   type_module_2 := 661;
   adr_module_2 := 25;
   bussystem_mod_2 := 1;
   bussystem_mod_3 := 1;
   bussystem_mod_4 := 1;
   slaveConfigInfo := DW#16#3;
   init_fb_done := DW#16#3;
   upload_done := DW#16#3;
   download_done := DW#16#3;
   cmdCtrl_FB37 := W#16#FE00;
   comCountStart_1 := W#16#2;
   mod_type_1 := W#16#1A17;
   mod_version_1 := W#16#3;
   dsv_info_mod_1 := W#16#1A3A;
   data_0_mod_1 := W#16#4545;
   data_2_mod_1 := W#16#10CC;
   data_4_mod_1 := W#16#20CC;
   data_6_mod_1 := W#16#203;
   data_8_mod_1 := W#16#F432;
   data_10_mod_1 := W#16#6400;
   data_12_mod_1 := W#16#6400;
   data_16_mod_1 := W#16#C00;
   data_18_mod_1 := W#16#2222;
   data_20_mod_1 := W#16#3A1A;
   data_22_mod_1 := W#16#FEFF;
   data_24_mod_1 := W#16#1E62;
   data_26_mod_1 := W#16#1F5B;
   data_30_mod_1 := W#16#7169;
   comCountStart_2 := W#16#2;
   mod_type_2 := W#16#19DB;
   mod_version_2 := W#16#3;
   dsv_info_mod_2 := W#16#4FA5;
   data_0_mod_2 := W#16#4545;
   data_2_mod_2 := W#16#10CC;
   data_4_mod_2 := W#16#20CC;
   data_6_mod_2 := W#16#201;
   data_8_mod_2 := W#16#421;
   data_10_mod_2 := W#16#6400;
   data_12_mod_2 := W#16#6400;
   data_16_mod_2 := W#16#A54F;
   data_18_mod_2 := W#16#FEFF;
   data_20_mod_2 := W#16#3E4E;
   data_22_mod_2 := W#16#735B;
   data_26_mod_2 := W#16#5953;
END_DATA_BLOCK

ORGANIZATION_BLOCK "Cycle"	// OB 1
TITLE = "Main Program Sweep (Cycle)"
AUTHOR : Koenig
VERSION : 0.1
VAR_TEMP
  OB1_EV_CLASS : BYTE ;	//Bits 0-3 = 1 (Coming event), Bits 4-7 = 1 (Event class 1)
  OB1_SCAN_1 : BYTE ;	//1 (Cold restart scan 1 of OB 1), 3 (Scan 2-n of OB 1)
  OB1_PRIORITY : BYTE ;	//Priority of OB Execution
  OB1_OB_NUMBR : BYTE ;	//1 (Organization block 1, OB1)
  OB1_RESERVED_1 : BYTE ;	//Reserved for system
  OB1_RESERVED_2 : BYTE ;	//Reserved for system
  OB1_PREV_CYCLE : INT ;	//Cycle time of previous OB1 scan (milliseconds)
  OB1_MIN_CYCLE : INT ;	//Minimum cycle time of OB1 (milliseconds)
  OB1_MAX_CYCLE : INT ;	//Maximum cycle time of OB1 (milliseconds)
  OB1_DATE_TIME : DATE_AND_TIME ;	//Date and time OB1 started
END_VAR
BEGIN
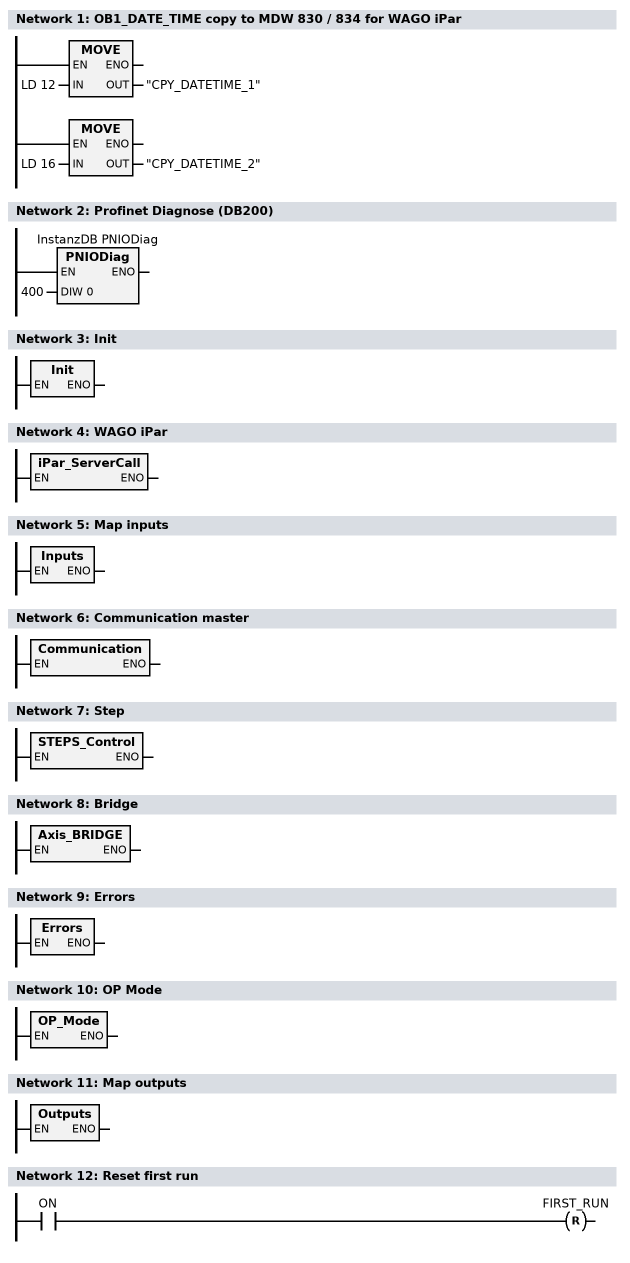
NETWORK
TITLE = OB1_DATE_TIME copy to MDW 830 / 834 for WAGO iPar
      L     LD 12;
      T     "CPY_DATETIME_1";
      L     LD 16;
      T     "CPY_DATETIME_2";
NETWORK
TITLE = Profinet Diagnose (DB200)
      CALL  "PNIODiag" , "InstanzDB PNIODiag" (
           DIW 0                    := 400);
      NOP   0;
NETWORK
TITLE = Init
      CALL  "Init";
      NOP   0;
NETWORK
TITLE = WAGO iPar
      CALL  "iPar_ServerCall";
      NOP   0;
NETWORK
TITLE = Map inputs
      CALL  "Inputs";
      NOP   0;
NETWORK
TITLE = Communication master
      CALL  "Communication";
      NOP   0;
NETWORK
TITLE = Step
      CALL  "STEPS_Control";
      NOP   0;
NETWORK
TITLE = Bridge
      CALL  "Axis_BRIDGE";
      NOP   0;
NETWORK
TITLE = Errors
      CALL  "Errors";
      NOP   0;
NETWORK
TITLE = OP Mode
      CALL  "OP_Mode";
      NOP   0;
NETWORK
TITLE = Map outputs
      CALL  "Outputs";
      NOP   0;
NETWORK
TITLE = Reset first run
      A     "ON";
      R     "FIRST_RUN";
END_ORGANIZATION_BLOCK

ORGANIZATION_BLOCK "CYC_INT5"	// OB 35
TITLE = "Cyclic Interrupt"
AUTHOR : Koenig
VERSION : 0.1
VAR_TEMP
  OB35_EV_CLASS : BYTE ;	//Bits 0-3 = 1 (Coming event), Bits 4-7 = 1 (Event class 1)
  OB35_STRT_INF : BYTE ;	//16#36 (OB 35 has started)
  OB35_PRIORITY : BYTE ;	//Priority of OB Execution
  OB35_OB_NUMBR : BYTE ;	//35 (Organization block 35, OB35)
  OB35_RESERVED_1 : BYTE ;	//Reserved for system
  OB35_RESERVED_2 : BYTE ;	//Reserved for system
  OB35_PHASE_OFFSET : WORD ;	//Phase offset (msec)
  OB35_RESERVED_3 : INT ;	//Reserved for system
  OB35_EXC_FREQ : INT ;	//Frequency of execution (msec)
  OB35_DATE_TIME : DATE_AND_TIME ;	//Date and time OB35 started
END_VAR
BEGIN
NETWORK
TITLE =
      CALL  "F-CALL";
END_ORGANIZATION_BLOCK

ORGANIZATION_BLOCK "I/O_FLT1"	// OB 82
TITLE = "I/O Point Fault"
AUTHOR : Koenig
VERSION : 0.1
VAR_TEMP
  OB82_EV_CLASS : BYTE ;	//16#39, Event class 3, Entering event state, Internal fault event
  OB82_FLT_ID : BYTE ;	//16#XX, Fault identifcation code
  OB82_PRIORITY : BYTE ;	//Priority of OB Execution
  OB82_OB_NUMBR : BYTE ;	//82 (Organization block 82, OB82)
  OB82_RESERVED_1 : BYTE ;	//Reserved for system
  OB82_IO_FLAG : BYTE ;	//Input (01010100), Output (01010101)
  OB82_MDL_ADDR : WORD ;	//Base address of module with fault
  OB82_MDL_DEFECT : BOOL ;	//Module defective
  OB82_INT_FAULT : BOOL ;	//Internal fault
  OB82_EXT_FAULT : BOOL ;	//External fault
  OB82_PNT_INFO : BOOL ;	//Point information
  OB82_EXT_VOLTAGE : BOOL ;	//External voltage low
  OB82_FLD_CONNCTR : BOOL ;	//Field wiring connector missing
  OB82_NO_CONFIG : BOOL ;	//Module has no configuration data
  OB82_CONFIG_ERR : BOOL ;	//Module has configuration error
  OB82_MDL_TYPE : BYTE ;	//Type of module
  OB82_SUB_MDL_ERR : BOOL ;	//Sub-Module is missing or has error
  OB82_COMM_FAULT : BOOL ;	//Communication fault
  OB82_MDL_STOP : BOOL ;	//Module is stopped
  OB82_WTCH_DOG_FLT : BOOL ;	//Watch dog timer stopped module
  OB82_INT_PS_FLT : BOOL ;	//Internal power supply fault
  OB82_PRIM_BATT_FLT : BOOL ;	//Primary battery is in fault
  OB82_BCKUP_BATT_FLT : BOOL ;	//Backup battery is in fault
  OB82_RESERVED_2 : BOOL ;	//Reserved for system
  OB82_RACK_FLT : BOOL ;	//Rack fault, only for bus interface module
  OB82_PROC_FLT : BOOL ;	//Processor fault
  OB82_EPROM_FLT : BOOL ;	//EPROM fault
  OB82_RAM_FLT : BOOL ;	//RAM fault
  OB82_ADU_FLT : BOOL ;	//ADU fault
  OB82_FUSE_FLT : BOOL ;	//Fuse fault
  OB82_HW_INTR_FLT : BOOL ;	//Hardware interupt input in fault
  OB82_RESERVED_3 : BOOL ;	//Reserved for system
  OB82_DATE_TIME : DATE_AND_TIME ;	//Date and time OB82 started
END_VAR
BEGIN
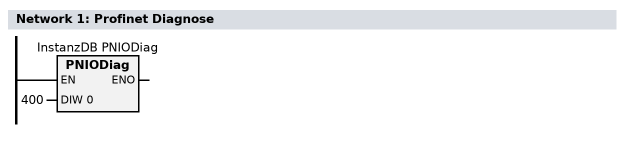
NETWORK
TITLE = Profinet Diagnose
      CALL  "PNIODiag" , "InstanzDB PNIODiag" (
           DIW 0                    := 400);
      NOP   0;
END_ORGANIZATION_BLOCK

ORGANIZATION_BLOCK "I/O_FLT2"	// OB 83
TITLE = "I/O Point Fault"
AUTHOR : Koenig
VERSION : 0.1
VAR_TEMP
  OB83_EV_CLASS : BYTE ;	//16#38/39, Event class 3, module inserted/removed (8/9)
  OB83_FLT_ID : BYTE ;	//16#XX, Fault identifcation code
  OB83_PRIORITY : BYTE ;	//Priority of OB Execution
  OB83_OB_NUMBR : BYTE ;	//83 (Organization block 83, OB83)
  OB83_RESERVED_1 : BYTE ;	//Reserved for system
  OB83_MDL_ID : BYTE ;	//Input module (01010100), Output module (01010101)
  OB83_MDL_ADDR : WORD ;	//Base address of module with point fault
  OB83_RACK_NUM : INT ;	//Number of rack that has module with point fault
  OB83_MDL_TYPE : WORD ;	//Module type with point fault
  OB83_DATE_TIME : DATE_AND_TIME ;	//Date and time OB83 started
END_VAR
BEGIN
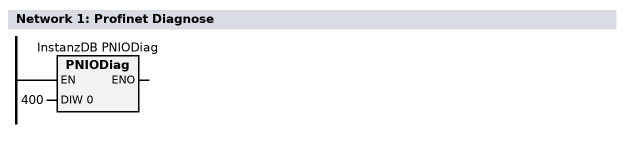
NETWORK
TITLE = Profinet Diagnose
      CALL  "PNIODiag" , "InstanzDB PNIODiag" (
           DIW 0                    := 400);
      NOP   0;
END_ORGANIZATION_BLOCK

ORGANIZATION_BLOCK "OBNL_FLT"	// OB 85
TITLE = "Organization Block (OB) Not Loaded Fault"
AUTHOR : Koenig
VERSION : 0.1
VAR_TEMP
  OB85_EV_CLASS : BYTE ;	//16#35 Event class 3
  OB85_FLT_ID : BYTE ;	//16#XX, Fault identification code
  OB85_PRIORITY : BYTE ;	//Priority of OB Execution
  OB85_OB_NUMBR : BYTE ;	//85 (Organization block 85, OB85)
  OB85_RESERVED_1 : BYTE ;	//Reserved for system
  OB85_RESERVED_2 : BYTE ;	//Reserved for system
  OB85_RESERVED_3 : INT ;	//Reserved for system
  OB85_ERR_EV_CLASS : BYTE ;	//Class of event causing error
  OB85_ERR_EV_NUM : BYTE ;	//Number of event causing error
  OB85_OB_PRIOR : BYTE ;	//Priority of OB causing error
  OB85_OB_NUM : BYTE ;	//Number of OB causing error
  OB85_DATE_TIME : DATE_AND_TIME ;	//Date and time OB85 started
END_VAR
BEGIN
NETWORK
TITLE =
END_ORGANIZATION_BLOCK

ORGANIZATION_BLOCK "RACK_FLT"	// OB 86
TITLE = "Loss Of Rack Fault"
AUTHOR : Koenig
VERSION : 0.1
VAR_TEMP
  OB86_EV_CLASS : BYTE ;	//16#38/39 Event class 3
  OB86_FLT_ID : BYTE ;	//16#C1/C4/C5, Fault identifcation code
  OB86_PRIORITY : BYTE ;	//Priority of OB Execution
  OB86_OB_NUMBR : BYTE ;	//86 (Organization block 86, OB86)
  OB86_RESERVED_1 : BYTE ;	//Reserved for system
  OB86_RESERVED_2 : BYTE ;	//Reserved for system
  OB86_MDL_ADDR : WORD ;	//Base address of IM module in rack with fault
  OB86_RACKS_FLTD : ARRAY  [0 .. 31 ] OF BOOL ;	//Racks in fault
  OB86_DATE_TIME : DATE_AND_TIME ;	//Date and time OB86 started
END_VAR
BEGIN
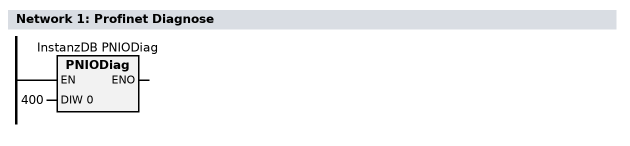
NETWORK
TITLE = Profinet Diagnose
      CALL  "PNIODiag" , "InstanzDB PNIODiag" (
           DIW 0                    := 400);
      NOP   0;
END_ORGANIZATION_BLOCK

ORGANIZATION_BLOCK "COMM_FLT"	// OB 87
TITLE = "Communication Fault"
AUTHOR : Koenig
VERSION : 0.1
VAR_TEMP
  OB87_EV_CLASS : BYTE ;	//16#39 Event class 3
  OB87_FLT_ID : BYTE ;	//16#XX, Fault identifcation code
  OB87_PRIORITY : BYTE ;	//Priority of OB Execution
  OB87_OB_NUMBR : BYTE ;	//87 (Organization block 87, OB87)
  OB87_RESERVED_1 : BYTE ;	//Reserved for system
  OB87_RESERVED_2 : BYTE ;	//Reserved for system
  OB87_RESERVED_3 : WORD ;	//Reserved for system
  OB87_RESERVED_4 : DWORD ;	//Reserved for system
  OB87_DATE_TIME : DATE_AND_TIME ;	//Date and time OB87 started
END_VAR
BEGIN
NETWORK
TITLE =
END_ORGANIZATION_BLOCK

ORGANIZATION_BLOCK "STARTUP"	// OB 100
TITLE = "Complete Restart"
AUTHOR : Koenig
VERSION : 0.1
VAR_TEMP
  OB100_EV_CLASS : BYTE ;	//16#13, Event class 1, Entering event state, Event logged in diagnostic buffer
  OB100_STRTUP : BYTE ;	//16#81/82/83/84 Method of startup
  OB100_PRIORITY : BYTE ;	//Priority of OB Execution
  OB100_OB_NUMBR : BYTE ;	//100 (Organization block 100, OB100)
  OB100_RESERVED_1 : BYTE ;	//Reserved for system
  OB100_RESERVED_2 : BYTE ;	//Reserved for system
  OB100_STOP : WORD ;	//Event that caused CPU to stop (16#4xxx)
  OB100_STRT_INFO : DWORD ;	//Information on how system started
  OB100_DATE_TIME : DATE_AND_TIME ;	//Date and time OB100 started
  ZeroDouble : DINT ;
  ret : INT ;
END_VAR
BEGIN
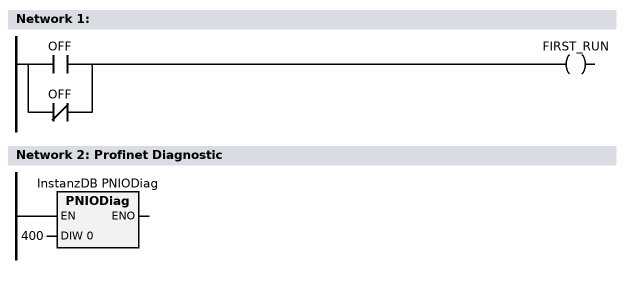
NETWORK
TITLE =
      O     "OFF";
      ON    "OFF";
      =     "FIRST_RUN";
NETWORK
TITLE = Profinet Diagnostic
      CALL  "PNIODiag" , "InstanzDB PNIODiag" (
           DIW 0                    := 400);
      NOP   0;
END_ORGANIZATION_BLOCK

ORGANIZATION_BLOCK "PROG_ERR"	// OB 121
TITLE = "Programming Error"
AUTHOR : Koenig
VERSION : 0.1
VAR_TEMP
  OB121_EV_CLASS : BYTE ;	//16#25, Event class 2, Entering event state, Internal fault event
  OB121_SW_FLT : BYTE ;	//16#XX Software programming fault
  OB121_PRIORITY : BYTE ;	//Priority of OB Execution
  OB121_OB_NUMBR : BYTE ;	//121 (Organization block 121, OB121)
  OB121_BLK_TYPE : BYTE ;	//16#88/8A/8B/8C/8E Type of block fault occured in
  OB121_RESERVED_1 : BYTE ;	//Reserved for system
  OB121_FLT_REG : WORD ;	//16#XX Specific register that caused fault
  OB121_BLK_NUM : WORD ;	//Number of block that programming fault occured in
  OB121_PRG_ADDR : WORD ;	//Address in block where programming fault occured
  OB121_DATE_TIME : DATE_AND_TIME ;	//Date and time OB121 started
END_VAR
BEGIN
NETWORK
TITLE =
END_ORGANIZATION_BLOCK

